// TIA Portal V16 program export: 21 tag tables, 13 data types, 28 data blocks, 76 code blocks (in call order from the OBs), 69 instance data blocks

VAR_GLOBAL   // PLC tag table "Default tag table"
   System_Byte AT %MB1 : Byte;
   FirstScan AT %M1.0 : Bool;
   DiagStatusUpdate AT %M1.1 : Bool;
   AlwaysTRUE AT %M1.2 : Bool;
   AlwaysFALSE AT %M1.3 : Bool;
   Clock_Byte AT %MB0 : Byte;
   Clock_10Hz AT %M0.0 : Bool;
   Clock_5Hz AT %M0.1 : Bool;
   "Clock_2.5Hz" AT %M0.2 : Bool;
   Clock_2Hz AT %M0.3 : Bool;
   "Clock_1.25Hz" AT %M0.4 : Bool;
   Clock_1Hz AT %M0.5 : Bool;
   "Clock_0.625Hz" AT %M0.6 : Bool;
   "Clock_0.5Hz" AT %M0.7 : Bool;
   trig_ustaw_czas AT %M206.1 : Bool;
   trig_pobierz_czas AT %M206.3 : Bool;
   "Bit_6-Wekt-Valve01_R" AT %M2000.6 : Bool;   // Bit-6 kasowanie alarmu
   "Bit_7-Wekt-Valve01_R" AT %M2000.7 : Bool;   // Bit trybu pracy napędu
   "Bit_5-Wekt-Valve01_R" AT %M2000.5 : Bool;   // Rozkaz zamykania
   "Bit_4-Wek_Valve01_R" AT %M2000.4 : Bool;   // Rozkaz otwieranie
   "Bit_0-Wekt_Valve01_R" AT %M2000.0 : Bool;   // Bit gotowośći / awarii
   "Bit_0-Wekt_Valve01_L" AT %M2001.0 : Bool;   // Bit Alarm/Gotowość (Alarm-=1, gotowość=0)
   "Bit_1-Wekt_Valve01_L" AT %M2001.1 : Bool;   // Bit potwierdzenia otwarcia
   "Bit_2-Wekt_Valve01_L" AT %M2001.2 : Bool;   // Bit wyboru trybu Zdalne=1 Remontowe=0
   "Bit_3-Wek_Valve01_L" AT %M2001.3 : Bool;   // Bit potwierdzenia zamknięcia
   "Bit_4-Wek_Valve01_L" AT %M2001.4 : Bool;   // Bit rozkazu na otwieranie
   "Bit_5-Wekt-Valve01_L" AT %M2001.5 : Bool;   // Bit rozkazu na zamykanie
   "Bit_6-Wekt-Valve01_L" AT %M2001.6 : Bool;   // Bit kasowania
   "Bit_7-Wekt-Valve01_L" AT %M2001.7 : Bool;   // Bit rodzaju sterowania aut =1 /manual= 0
   Byte_Wekt_Valve01_L AT %MB2001 : Byte;   // Lewy byte wektora napędu
   Byte_Wekt_Valve01_R AT %MB2000 : Byte;   // Prawy byte wektora napędu
   "I0.3" AT %I0.3 : Bool;
   "I0.4" AT %I0.4 : Bool;
   "I0.5" AT %I0.5 : Bool;
   "I0.6" AT %I0.6 : Bool;
   "Q0.3" AT %Q0.3 : Bool;
   "Q0.4" AT %Q0.4 : Bool;
   "Q0.5" AT %Q0.5 : Bool;
   "I6.4" AT %I6.4 : Bool;
   "I6.3" AT %I6.3 : Bool;
   "I6.2" AT %I6.2 : Bool;
   "I9.5" AT %I9.5 : Bool;
   "I9.6" AT %I9.6 : Bool;
   "I9.7" AT %I9.7 : Bool;
   "I3.1" AT %I3.1 : Bool;
   "I3.2" AT %I3.2 : Bool;
   "I3.3" AT %I3.3 : Bool;
   "I3.4" AT %I3.4 : Bool;
   "Q2.5" AT %Q2.5 : Bool;
   "Q2.6" AT %Q2.6 : Bool;
   "Q2.7" AT %Q2.7 : Bool;
   "I6.1" AT %I6.1 : Bool;
   "Bit_1-Wekt_Valve01_R" AT %M2000.1 : Bool;   // Bit potwierdzenia otwarcia
   "Byte_Wekt_POSITION_R(1)" AT %MB2002 : Byte;   // Prawy byte wektora napędu
   "Bit_0-Wekt_POSITION_R(1)" AT %M2002.0 : Bool;   // Bit gotowośći / awarii
   "Bit_1-Wekt_POSITION_R(1)" AT %M2002.1 : Bool;   // Bit potwierdzenia otwarcia
   "Bit_4-Wek_POSITION_R(1)" AT %M2002.4 : Bool;   // Rozkaz otwieranie
   "Bit_5-Wekt_POSITION_R(1)" AT %M2002.5 : Bool;   // Rozkaz zamykania
   "Bit_6-Wekt_POSITION_R(1)" AT %M2002.6 : Bool;   // Bit-6 kasowanie alarmu
   "Bit_7-Wekt_POSITION_R(1)" AT %M2002.7 : Bool;   // Bit trybu pracy napędu
   "Byte_Wekt_POSITION_L(1)" AT %MB2003 : Byte;   // Lewy byte wektora napędu
   "Bit_0-Wekt_POSITION_L(1)" AT %M2003.0 : Bool;   // Bit Alarm/Gotowość (Alarm-=1, gotowość=0)
   "Bit_1-Wekt_POSITION_L(1)" AT %M2003.1 : Bool;   // Bit potwierdzenia otwarcia
   "Bit_2-Wekt_POSITION_L(1)" AT %M2003.2 : Bool;   // Bit wyboru trybu Zdalne=1 Remontowe=0
   "Bit_3-Wek_POSITION_L(1)" AT %M2003.3 : Bool;   // Bit potwierdzenia zamknięcia
   "Bit_4-Wek_POSITION_L(1)" AT %M2003.4 : Bool;   // Bit rozkazu na otwieranie
   "Bit_5-Wekt_POSITION_L(1)" AT %M2003.5 : Bool;   // Bit rozkazu na zamykanie
   "Bit_6-Wekt_POSITION_L(1)" AT %M2003.6 : Bool;   // Bit kasowania
   "Bit_7-Wekt_POSITION_L(1)" AT %M2003.7 : Bool;   // Bit rodzaju sterowania aut =1 /manual= 0
   "Bit_2-Wekt_POSITION_R(1)" AT %M2002.2 : Bool;   // Bit wyboru trybu Zdalne=1 Remontowe=0
   "Bit_3-Wek_POSITION_R(1)" AT %M2002.3 : Bool;   // Bit potwierdzenia zamknięcia
   Tag_1 AT %M5000.0 : Bool;
   Tag_2 AT %M5000.1 : Bool;
   Tag_3 AT %M5000.3 : Bool;
   "I3.6" AT %I3.6 : Bool;
   "I3.7" AT %I3.7 : Bool;
   "I4.0" AT %I4.0 : Bool;
   "I3.5" AT %I3.5 : Bool;
   "I6.7" AT %I6.7 : Bool;
   "I6.6" AT %I6.6 : Bool;
   "I6.5" AT %I6.5 : Bool;
   "Q3.0" AT %Q3.0 : Bool;
   "Q3.1" AT %Q3.1 : Bool;
   "Q3.2" AT %Q3.2 : Bool;
   My_1Hz AT %M206.7 : Bool;
   "I1.1" AT %I1.1 : Bool;
   "I0.7" AT %I0.7 : Bool;
   "I1.0" AT %I1.0 : Bool;
   "I1.2" AT %I1.2 : Bool;
   "I7.0" AT %I7.0 : Bool;
   "I7.1" AT %I71.1 : Bool;
   "I7.2" AT %I7.2 : Bool;
   "Q3.4" AT %Q3.4 : Bool;
   "Q3.5" AT %Q3.5 : Bool;
   "Q3.6" AT %Q3.6 : Bool;
   "Q1.1" AT %Q1.1 : Bool;
   "Q2.0" AT %Q2.0 : Bool;
   "Q2.1" AT %Q2.1 : Bool;
   "I1.3" AT %I1.3 : Bool;
   "I1.4" AT %I1.4 : Bool;
   "I1.5" AT %I1.5 : Bool;
   "I2.0" AT %I2.0 : Bool;
   "I7.6" AT %I7.6 : Bool;
   "I7.7" AT %I7.7 : Bool;
   "I8.0" AT %I8.0 : Bool;
   "I7.3" AT %I7.3 : Bool;
   "I7.4" AT %I7.4 : Bool;
   "I7.5" AT %I7.5 : Bool;
   "I4.1" AT %I4.1 : Bool;
   "I4.2" AT %I4.2 : Bool;
   "I4.3" AT %I4.3 : Bool;
   "I4.4" AT %I4.4 : Bool;
   "I8.1" AT %I8.1 : Bool;
   "I8.2" AT %I8.2 : Bool;
   "I8.3" AT %I8.3 : Bool;
   "I4.5" AT %I4.5 : Bool;
   "I4.6" AT %I4.6 : Bool;
   "I4.7" AT %I4.7 : Bool;
   "I5.0" AT %I5.0 : Bool;
   "Q3.7" AT %Q3.7 : Bool;
   "Q4.0" AT %Q4.0 : Bool;
   "Q4.1" AT %Q4.1 : Bool;
   "Q2.2" AT %Q2.2 : Bool;
   "Q2.3" AT %Q2.3 : Bool;
   "Q2.4" AT %Q2.4 : Bool;
   "I2.1" AT %I2.1 : Bool;
   "I2.2" AT %I2.2 : Bool;
   "I2.3" AT %I2.3 : Bool;
   "I2.4" AT %I2.4 : Bool;
   "I8.4" AT %I8.4 : Bool;
   "I8.5" AT %I8.5 : Bool;
   "I8.6" AT %I8.6 : Bool;
   "I8.7" AT %I8.7 : Bool;
   "I9.0" AT %I9.0 : Bool;
   "I9.1" AT %I9.1 : Bool;
   "I5.1" AT %I5.1 : Bool;
   "I5.2" AT %I5.2 : Bool;
   "I5.3" AT %I5.3 : Bool;
   "I5.4" AT %I5.4 : Bool;
   "Q4.2" AT %Q4.2 : Bool;
   "Q4.3" AT %Q4.3 : Bool;
   "Q4.4" AT %Q4.4 : Bool;
   "I9.2" AT %I9.2 : Bool;
   "I9.3" AT %I9.3 : Bool;
   "I9.4" AT %I9.4 : Bool;
   "I0.0" AT %I0.0 : Bool;
   "I0.1" AT %I0.1 : Bool;
   "I0.2" AT %I0.2 : Bool;
   "Q0.6" AT %Q0.6 : Bool;
   "Q0.7" AT %Q0.7 : Bool;
   "Q1.0" AT %Q1.0 : Bool;
   "Q0.0" AT %Q0.0 : Bool;
   "Q0.1" AT %Q0.1 : Bool;
   "Q0.2" AT %Q0.2 : Bool;
   "I10.0" AT %I10.0 : Bool;
   setTime AT %M8.0 : Bool;   // ustaw zegar
   setData AT %M8.1 : Bool;   // ustaw datę
   isDaily AT %M80.7 : Bool;   // tryb sterowania dobowy
   isWeekiy AT %M81.0 : Bool;   // tryb sterowania tygodniowy
   isPowerOK AT %M81.2 : Bool;   // znacznik powrotu zasilania
   Tag_4 AT %Q6.7 : Bool;
   zbocze_dod_zegar AT %M47.0 : Bool;
   ResetErrorOB82 AT %M91.1 : Bool;
   "I5.5" AT %I5.5 : Bool;
   "I5.6" AT %I5.6 : Bool;
   "I5.7" AT %I5.7 : Bool;
   "I6.0" AT %I6.0 : Bool;
END_VAR
VAR_GLOBAL CONSTANT   // user constants
   analog_error_H : Word := 28538;
   CONST_BUFFER_OB82 : USInt := 200;
END_VAR

VAR_GLOBAL   // PLC tag table "Alarm_error"
   errorAnlog_Z10 AT %M9.3 : Bool;   // sygnał błędu sygnału analogowego położenia Z10
   outAlarm AT %M1030.3 : Bool;   // Znacznik alarmu zbiorczego (Sygnalizator)
   float_min_tank_4 AT %M47.4 : Bool;   // pływak min zbiornik 4
   float_min_tank_1 AT %M47.1 : Bool;   // pływak min zbiornik 1
   float_min_tank_3 AT %M47.3 : Bool;   // pływak min zbiornik 3
   float_min_tank_2 AT %M47.2 : Bool;   // pływak min zbiornik 2
   "I2.7" AT %I2.7 : Bool;
   "I3.0" AT %I3.0 : Bool;
   "I2.6" AT %I2.6 : Bool;
   "I2.5" AT %I2.5 : Bool;
   Communication_alarm_tcp AT %M1030.2 : Bool;   // Znacznik błedu komunikacji HMI - PLC
   comunication_alarm_modbus_rtu AT %M1030.4 : Bool;   // kontrola przebiegu pętli odczytu parametró z modbus rtu
   Led_Error AT %M91.0 : Bool;   // bit sygnalizacji zapalenia led error na CPU
   Status_QRY AT %MW302 : Word;   // Status słowa przerwań (bit 0 - informacja o CPU 0- RUN, 1- Rozruch)
   statusCPU AT %M302.0 : Bool;   // 0- Run 1-Rozruch
   Error_QRY AT %MW300 : Int;   // Słowo błędu przetwarzania przerwań czasowych
   setAlarmNiskie_magistrala AT %M91.2 : Bool;   // bit alarmu niskiego ciśnienia na magistrali
   resetAlarmNiskie_magistrala AT %M91.3 : Bool;   // bit końca niskiego ciśnienia magistrala
   float_max_tank_3 AT %M46.6 : Bool;   // pływak max zbiornik 3
   float_max_tank_1 AT %M46.4 : Bool;   // pływak max zbiornik 1
   setControl_alarm_B5 AT %M91.4 : Bool;   // Załczenie sterowania zbiornikami w trybie awarii na magistrali
   float_max_tank_2 AT %M46.5 : Bool;   // pływak max zbiornik 2
   float_max_tank_4 AT %M46.7 : Bool;   // pływak max zbiornik 2
   reset_error_hwork AT %M45.6 : Bool;   // reset po błędzie gdy wszystkie zbiorniki ten sam czas pracy
END_VAR

VAR_GLOBAL   // PLC tag table "Analogi"
   AI_poziom_zbiornik_4 AT %MW42 : Word;
   AI_poziom_zbiornik_2 AT %MW38 : Word;
   IW68 AT %IW68 : Word;   // wejscie AI
   AI_poziom_zbiornik_1 AT %MW36 : Word;
   AI_poziom_zbiornik_3 AT %MW40 : Word;
   IW78 AT %IW78 : Word;   // wejscie AI
   AI_położenie_Z10 AT %MW34 : Word;
   AI_przepływ AT %MW30 : Word;
   AI_ciśnienie_B5 AT %MW32 : Word;
   IW70 AT %IW70 : Word;   // wejscie AI
   IW72 AT %IW72 : Word;   // wejscie AI
   IW76 AT %IW76 : Word;   // wejscie AI
   IW74 AT %IW74 : Word;   // wejscie AI
   switch_Kolman AT %M46.0 : Bool;   // przełącznik funkcji filtr analogów (Kolman = OFF, bez Kolman = ON)
   I AT %MW48 : Int;   // kalman zmienna przechwuje adres wejścia AI
END_VAR

VAR_GLOBAL   // PLC tag table "Tag HMI"
   "HMI.ManualMode_visible" AT %M1023.1 : Bool;
   "HMI.ErrorBits_Int" AT %MW1024 : Int;
   "HMI.Warning_Int" AT %MW1028 : Int;
   "HMI.ErrorAck_Int" AT %MW1026 : Int;
   ProcessMemory_Static_1_setChanging AT %M9.2 : Bool;   // Znacznik pobierania konfiguracji do instancji pamięci peocesu
   "HMI.Acknowledge_visible" AT %M1030.1 : Bool;
   memRis_WatchDog_HMI_PLC AT %M9.0 : Bool;
   "HMI.ErrorAck" AT %M1030.0 : Bool;
   "HMI.Filing3" AT %M1031.4 : Bool;   // bit informujący o wejściu w tryb napełniania
   "HMI.Warning_Int_tank" AT %MW1031 : Int;
   "HMI.rez" AT %M1031.1 : Bool;
   "HMI.StopFiling" AT %M1031.0 : Bool;   // bit informacji o zatrzymanym napełnianiu z powodu niskiego ciśnienia wna magistrali
   "HMI.Filing2" AT %M1031.3 : Bool;   // bit informujący o wejściu w tryb napełniania
   "HMI.Filing4" AT %M1031.5 : Bool;   // bit informujący o wejściu w tryb napełniania
   "HMI.Filing1" AT %M1031.2 : Bool;   // bit informujący o wejściu w tryb napełniania
END_VAR

VAR_GLOBAL   // PLC tag table "ModbusRTU"
   switch_flow_analog_modbus AT %M79.0 : Bool;   // przełącznik wyboru medium pomiaru przepływu z wy analogowego czy modbus rtu
END_VAR

VAR_GLOBAL   // PLC tag table "ModbusTCP"
   memTrig_Client_ReceivingTIME AT %M206.4 : Bool;
   memTrig_Step_Sending AT %M9.4 : Bool;   // Pamieć zbocza na uruchomienie pętli Modbus TCP wysyłanie
   done_modbusTCP_przetworzone AT %M9.1 : Bool;   // bit zezwala na wysłanie danych po przetworzeniu przez program PLC Zasuwy
   memTrig_Step_Receiving_Time AT %M9.6 : Bool;   // Pamieć zbocza na uruchomienie pętli Modbus TCP pobieranie Time
   memTrig_Step_Receiving AT %M9.5 : Bool;   // Pamieć zbocza na uruchomienie pętli Modbus TCP pobieranie
   memRisingTriger_Data_13 AT %M208.4 : Bool;   // pamieć zbocza zmiany danych w zmiennej
   memRisingTriger_Data_9 AT %M208.0 : Bool;   // pamieć zbocza zmiany danych w zmiennej
   memRisingTriger_Data_6 AT %M207.5 : Bool;   // pamieć zbocza zmiany danych w zmiennej
   memRisingTriger_Data_5 AT %M207.4 : Bool;   // pamieć zbocza zmiany danych w zmiennej
   memRisingTriger_Data_7 AT %M207.6 : Bool;   // pamieć zbocza zmiany danych w zmiennej
   memRisingTriger_Data_10 AT %M208.1 : Bool;   // pamieć zbocza zmiany danych w zmiennej
   memRisingTriger_Data_8 AT %M207.7 : Bool;   // pamieć zbocza zmiany danych w zmiennej
   memRisingTriger_Data_11 AT %M208.2 : Bool;   // pamieć zbocza zmiany danych w zmiennej
   memRisingTriger_Data_1 AT %M207.0 : Bool;   // pamieć zbocza zmiany danych w zmiennej
   memRisingTriger_Data_2 AT %M207.1 : Bool;   // pamieć zbocza zmiany danych w zmiennej
   memRisingTriger_Data_4 AT %M207.3 : Bool;   // pamieć zbocza zmiany danych w zmiennej
   memRisingTriger_Data_12 AT %M208.3 : Bool;   // pamieć zbocza zmiany danych w zmiennej
   memRisingTriger_Data_3 AT %M207.2 : Bool;   // pamieć zbocza zmiany danych w zmiennej
   memRisingTriger_Data_1_2 AT %M212.4 : Bool;   // pamieć zbocza zmiany danych w zmiennej
   memTrig_SendingError_4 AT %M210.7 : Bool;   // bit pamęci zbocza błedu wysyłania modbus tCP
   memTrig_Client_Receiving_12 AT %M210.1 : Bool;   // pamieć zbocza zmiany danych w zmiennej
   memTrig_Client_Receiving_3 AT %M209.0 : Bool;   // pamieć zbocza zmiany danych w zmiennej
   memTrig_Client_Receiving_9 AT %M209.6 : Bool;   // pamieć zbocza zmiany danych w zmiennej
   memTrig_Client_Receiving_11 AT %M210.0 : Bool;   // pamieć zbocza zmiany danych w zmiennej
   memTrig_Step_Sending_1 AT %M211.0 : Bool;   // Pamieć zbocza na uruchomienie pętli Modbus TCP wysyłanie
   memTrig_Client_Receiving_6 AT %M209.3 : Bool;   // pamieć zbocza zmiany danych w zmiennej
   memTrig_Client_Receiving_4 AT %M209.1 : Bool;   // pamieć zbocza zmiany danych w zmiennej
   done_modbusTCP_przetw_1 AT %M211.1 : Bool;   // bit zezwala na wysłanie danych po przetworzeniu przez program PLC Zasuwy
   memTrig_SendingError_2 AT %M210.5 : Bool;   // bit pamęci zbocza błedu wysyłania modbus tCP
   done_modbusTCP_przetw_6 AT %M212.2 : Bool;   // bit zezwala na wysłanie danych po przetworzeniu przez program PLC Zasuwy
   memTrig_Client_Receiving_2 AT %M208.7 : Bool;   // pamieć zbocza zmiany danych w zmiennej
   done_modbusTCP_przetw_4 AT %M212.0 : Bool;   // bit zezwala na wysłanie danych po przetworzeniu przez program PLC Zasuwy
   done_modbusTCP_przetw_2 AT %M211.2 : Bool;   // bit zezwala na wysłanie danych po przetworzeniu przez program PLC Zasuwy
   memTrig_Client_Receiving_7 AT %M209.4 : Bool;   // pamieć zbocza zmiany danych w zmiennej
   memTrig_Client_Receiving_13 AT %M210.2 : Bool;   // pamieć zbocza zmiany danych w zmiennej
   memRisingTriger_Data_1_1 AT %M212.3 : Bool;   // pamieć zbocza zmiany danych w zmiennej
   memTrig_Client_Receiving_5 AT %M209.2 : Bool;   // pamieć zbocza zmiany danych w zmiennej
   memRisingTriger_Data_1_5 AT %M212.7 : Bool;   // pamieć zbocza zmiany danych w zmiennej
   memTrig_Client_Receiving_1 AT %M208.6 : Bool;   // pamieć zbocza zmiany danych w zmiennej
   memTrig_Step_Sending_4 AT %M211.6 : Bool;   // Pamieć zbocza na uruchomienie pętli Modbus TCP wysyłanie
   memTrig_Client_Receiving_10 AT %M209.7 : Bool;   // pamieć zbocza zmiany danych w zmiennej
   memRisingTriger_Data_1_4 AT %M212.6 : Bool;   // pamieć zbocza zmiany danych w zmiennej
   memTrig_Client_Receiving_8 AT %M209.5 : Bool;   // pamieć zbocza zmiany danych w zmiennej
   memTrig_SendingError_3 AT %M210.6 : Bool;   // bit pamęci zbocza błedu wysyłania modbus tCP
   memTrig_Step_Sending_5 AT %M211.7 : Bool;   // Pamieć zbocza na uruchomienie pętli Modbus TCP wysyłanie
   done_modbusTCP_przetw_3 AT %M211.3 : Bool;   // bit zezwala na wysłanie danych po przetworzeniu przez program PLC Zasuwy
   memRisingTriger_Data_1_3 AT %M212.5 : Bool;   // pamieć zbocza zmiany danych w zmiennej
   memTrig_Step_Sending_2 AT %M211.4 : Bool;   // Pamieć zbocza na uruchomienie pętli Modbus TCP wysyłanie
   done_modbusTCP_przetw_5 AT %M212.1 : Bool;   // bit zezwala na wysłanie danych po przetworzeniu przez program PLC Zasuwy
   memTrig_SendingError_1 AT %M210.4 : Bool;   // bit pamęci zbocza błedu wysyłania modbus tCP
   memTrig_Client_Receiving_14 AT %M210.3 : Bool;   // pamieć zbocza zmiany danych w zmiennej
   memTrig_Step_Sending_3 AT %M211.5 : Bool;   // Pamieć zbocza na uruchomienie pętli Modbus TCP wysyłanie
   memTrig_Error_Receiving AT %M208.5 : Bool;   // pamieć zboczawystąpienia błędu pobierania
   memRisingTriger_Data_16 AT %M213.2 : Bool;   // pamieć zbocza zmiany danych w zmiennej
   memTrig_Client_Receiving_15 AT %M213.3 : Bool;   // pamieć zbocza zmiany danych w zmiennej
   memRisingTriger_Data_14 AT %M213.0 : Bool;   // pamieć zbocza zmiany danych w zmiennej
   memTrig_Client_Receiving_16 AT %M213.4 : Bool;   // pamieć zbocza zmiany danych w zmiennej
   memRisingTriger_Data_15 AT %M213.1 : Bool;   // pamieć zbocza zmiany danych w zmiennej
   memTrig_loop_error AT %M206.5 : Bool;   // błąd petli Modbus TCP brak obiegu pętli
   memRisingTriger_Data_50 AT %M227.1 : Bool;
   memTrig_Client_Receiving_37 AT %M216.4 : Bool;   // pamieć zbocza zmiany danych w zmiennej
   memRisingTriger_Data_83 AT %M231.2 : Bool;
   memTrig_Client_Receiving_84 AT %M222.3 : Bool;   // pamieć zbocza zmiany danych w zmiennej
   memRisingTriger_Data_76 AT %M230.3 : Bool;
   memRisingTriger_Data_18 AT %M223.1 : Bool;
   memTrig_Client_Receiving_38 AT %M216.5 : Bool;   // pamieć zbocza zmiany danych w zmiennej
   memRisingTriger_Data_89 AT %M232.0 : Bool;
   memTrig_Client_Receiving_17 AT %M214.0 : Bool;   // pamieć zbocza zmiany danych w zmiennej
   memTrig_Client_Receiving_81 AT %M222.0 : Bool;   // pamieć zbocza zmiany danych w zmiennej
   memRisingTriger_Data_81 AT %M231.0 : Bool;
   memTrig_Client_Receiving_66 AT %M220.1 : Bool;   // pamieć zbocza zmiany danych w zmiennej
   memTrig_Client_Receiving_62 AT %M219.5 : Bool;   // pamieć zbocza zmiany danych w zmiennej
   memTrig_Client_Receiving_21 AT %M214.4 : Bool;   // pamieć zbocza zmiany danych w zmiennej
   memTrig_Client_Receiving_65 AT %M220.0 : Bool;   // pamieć zbocza zmiany danych w zmiennej
   memTrig_Client_Receiving_43 AT %M217.2 : Bool;   // pamieć zbocza zmiany danych w zmiennej
   memRisingTriger_Data_85 AT %M231.4 : Bool;
   memTrig_Client_Receiving_25 AT %M215.0 : Bool;   // pamieć zbocza zmiany danych w zmiennej
   memRisingTriger_Data_70 AT %M229.5 : Bool;
   memTrig_Client_Receiving_46 AT %M217.5 : Bool;   // pamieć zbocza zmiany danych w zmiennej
   memTrig_Client_Receiving_47 AT %M217.6 : Bool;   // pamieć zbocza zmiany danych w zmiennej
   memTrig_Client_Receiving_18 AT %M214.1 : Bool;   // pamieć zbocza zmiany danych w zmiennej
   memRisingTriger_Data_40 AT %M225.7 : Bool;
   memRisingTriger_Data_86 AT %M231.5 : Bool;
   memRisingTriger_Data_68 AT %M229.3 : Bool;
   memTrig_Client_Receiving_19 AT %M214.2 : Bool;   // pamieć zbocza zmiany danych w zmiennej
   memTrig_Client_Receiving_41 AT %M217.0 : Bool;   // pamieć zbocza zmiany danych w zmiennej
   memRisingTriger_Data_45 AT %M226.4 : Bool;
   memTrig_Client_Receiving_64 AT %M219.7 : Bool;   // pamieć zbocza zmiany danych w zmiennej
   memRisingTriger_Data_28 AT %M224.3 : Bool;
   memTrig_Client_Receiving_49 AT %M218.0 : Bool;   // pamieć zbocza zmiany danych w zmiennej
   memRisingTriger_Data_65 AT %M229.0 : Bool;
   memTrig_Client_Receiving_35 AT %M216.2 : Bool;   // pamieć zbocza zmiany danych w zmiennej
   memRisingTriger_Data_21 AT %M223.4 : Bool;
   memTrig_Client_Receiving_72 AT %M220.7 : Bool;   // pamieć zbocza zmiany danych w zmiennej
   memTrig_Client_Receiving_57 AT %M219.0 : Bool;   // pamieć zbocza zmiany danych w zmiennej
   memTrig_Client_Receiving_51 AT %M218.2 : Bool;   // pamieć zbocza zmiany danych w zmiennej
   memTrig_Client_Receiving_28 AT %M215.3 : Bool;   // pamieć zbocza zmiany danych w zmiennej
   memRisingTriger_Data_66 AT %M229.1 : Bool;
   memTrig_Client_Receiving_45 AT %M217.4 : Bool;   // pamieć zbocza zmiany danych w zmiennej
   memTrig_Client_Receiving_89 AT %M223.0 : Bool;   // pamieć zbocza zmiany danych w zmiennej
   memRisingTriger_Data_35 AT %M225.2 : Bool;
   memTrig_Client_Receiving_83 AT %M222.2 : Bool;   // pamieć zbocza zmiany danych w zmiennej
   memRisingTriger_Data_56 AT %M227.7 : Bool;
   memRisingTriger_Data_20 AT %M223.3 : Bool;
   memTrig_Client_Receiving_36 AT %M216.3 : Bool;   // pamieć zbocza zmiany danych w zmiennej
   memTrig_Client_Receiving_26 AT %M215.1 : Bool;   // pamieć zbocza zmiany danych w zmiennej
   memRisingTriger_Data_23 AT %M223.6 : Bool;
   memRisingTriger_Data_48 AT %M226.7 : Bool;
   memRisingTriger_Data_64 AT %M228.7 : Bool;
   memRisingTriger_Data_61 AT %M228.4 : Bool;
   memRisingTriger_Data_36 AT %M225.3 : Bool;
   memRisingTriger_Data_88 AT %M231.7 : Bool;
   memTrig_Client_Receiving_76 AT %M221.3 : Bool;   // pamieć zbocza zmiany danych w zmiennej
   memRisingTriger_Data_72 AT %M229.7 : Bool;
   memRisingTriger_Data_74 AT %M230.1 : Bool;
   memRisingTriger_Data_39 AT %M225.6 : Bool;
   memRisingTriger_Data_90 AT %M232.1 : Bool;
   memRisingTriger_Data_25 AT %M224.0 : Bool;
   memRisingTriger_Data_44 AT %M226.3 : Bool;
   memRisingTriger_Data_80 AT %M230.7 : Bool;
   memTrig_Client_Receiving_70 AT %M220.5 : Bool;   // pamieć zbocza zmiany danych w zmiennej
   memRisingTriger_Data_37 AT %M225.4 : Bool;
   memTrig_Client_Receiving_20 AT %M214.3 : Bool;   // pamieć zbocza zmiany danych w zmiennej
   memTrig_Client_Receiving_34 AT %M216.1 : Bool;   // pamieć zbocza zmiany danych w zmiennej
   memRisingTriger_Data_49 AT %M227.0 : Bool;
   memRisingTriger_Data_78 AT %M230.5 : Bool;
   memRisingTriger_Data_38 AT %M225.5 : Bool;
   memTrig_Client_Receiving_87 AT %M222.6 : Bool;   // pamieć zbocza zmiany danych w zmiennej
   memTrig_Client_Receiving_30 AT %M215.5 : Bool;   // pamieć zbocza zmiany danych w zmiennej
   memRisingTriger_Data_42 AT %M226.1 : Bool;
   memRisingTriger_Data_57 AT %M228.0 : Bool;
   memTrig_Client_Receiving_54 AT %M218.5 : Bool;   // pamieć zbocza zmiany danych w zmiennej
   memRisingTriger_Data_77 AT %M230.4 : Bool;
   memTrig_Client_Receiving_86 AT %M222.5 : Bool;   // pamieć zbocza zmiany danych w zmiennej
   memTrig_Client_Receiving_63 AT %M219.6 : Bool;   // pamieć zbocza zmiany danych w zmiennej
   memTrig_Client_Receiving_67 AT %M220.2 : Bool;   // pamieć zbocza zmiany danych w zmiennej
   memTrig_Client_Receiving_75 AT %M221.2 : Bool;   // pamieć zbocza zmiany danych w zmiennej
   memRisingTriger_Data_54 AT %M227.5 : Bool;
   memTrig_Client_Receiving_24 AT %M214.7 : Bool;   // pamieć zbocza zmiany danych w zmiennej
   memRisingTriger_Data_41 AT %M226.0 : Bool;
   memTrig_Client_Receiving_82 AT %M222.1 : Bool;   // pamieć zbocza zmiany danych w zmiennej
   memRisingTriger_Data_75 AT %M230.2 : Bool;
   memTrig_Client_Receiving_61 AT %M219.4 : Bool;   // pamieć zbocza zmiany danych w zmiennej
   memRisingTriger_Data_59 AT %M228.2 : Bool;
   memRisingTriger_Data_33 AT %M225.0 : Bool;
   memRisingTriger_Data_19 AT %M223.2 : Bool;
   memTrig_Client_Receiving_56 AT %M218.7 : Bool;   // pamieć zbocza zmiany danych w zmiennej
   memTrig_Client_Receiving_88 AT %M222.7 : Bool;   // pamieć zbocza zmiany danych w zmiennej
   memRisingTriger_Data_47 AT %M226.6 : Bool;
   memTrig_Client_Receiving_59 AT %M219.2 : Bool;   // pamieć zbocza zmiany danych w zmiennej
   memTrig_Client_Receiving_48 AT %M217.7 : Bool;   // pamieć zbocza zmiany danych w zmiennej
   memTrig_Client_Receiving_23 AT %M214.6 : Bool;   // pamieć zbocza zmiany danych w zmiennej
   memTrig_Client_Receiving_32 AT %M215.7 : Bool;   // pamieć zbocza zmiany danych w zmiennej
   memTrig_Client_Receiving_53 AT %M218.4 : Bool;   // pamieć zbocza zmiany danych w zmiennej
   memRisingTriger_Data_79 AT %M230.6 : Bool;
   memRisingTriger_Data_43 AT %M226.2 : Bool;
   memRisingTriger_Data_73 AT %M230.0 : Bool;
   memRisingTriger_Data_87 AT %M231.6 : Bool;
   memRisingTriger_Data_58 AT %M228.1 : Bool;
   memRisingTriger_Data_69 AT %M229.4 : Bool;
   memTrig_Client_Receiving_42 AT %M217.1 : Bool;   // pamieć zbocza zmiany danych w zmiennej
   memTrig_Client_Receiving_69 AT %M220.4 : Bool;   // pamieć zbocza zmiany danych w zmiennej
   memTrig_Client_Receiving_44 AT %M217.3 : Bool;   // pamieć zbocza zmiany danych w zmiennej
   memTrig_Client_Receiving_85 AT %M222.4 : Bool;   // pamieć zbocza zmiany danych w zmiennej
   memTrig_Client_Receiving_31 AT %M215.6 : Bool;   // pamieć zbocza zmiany danych w zmiennej
   memTrig_Client_Receiving_27 AT %M215.2 : Bool;   // pamieć zbocza zmiany danych w zmiennej
   memRisingTriger_Data_24 AT %M223.7 : Bool;
   memTrig_Client_Receiving_50 AT %M218.1 : Bool;   // pamieć zbocza zmiany danych w zmiennej
   memRisingTriger_Data_17 AT %M206.6 : Bool;
   memTrig_Client_Receiving_22 AT %M214.5 : Bool;   // pamieć zbocza zmiany danych w zmiennej
   memRisingTriger_Data_52 AT %M227.3 : Bool;
   memRisingTriger_Data_55 AT %M227.6 : Bool;
   memRisingTriger_Data_34 AT %M225.1 : Bool;
   memTrig_Client_Receiving_77 AT %M221.4 : Bool;   // pamieć zbocza zmiany danych w zmiennej
   memRisingTriger_Data_82 AT %M231.1 : Bool;
   memRisingTriger_Data_67 AT %M229.2 : Bool;
   memRisingTriger_Data_26 AT %M224.1 : Bool;
   memTrig_Client_Receiving_60 AT %M219.3 : Bool;   // pamieć zbocza zmiany danych w zmiennej
   memRisingTriger_Data_27 AT %M224.2 : Bool;
   memTrig_Client_Receiving_52 AT %M218.3 : Bool;   // pamieć zbocza zmiany danych w zmiennej
   memRisingTriger_Data_84 AT %M231.3 : Bool;
   memTrig_Client_Receiving_29 AT %M215.4 : Bool;   // pamieć zbocza zmiany danych w zmiennej
   memTrig_Client_Receiving_73 AT %M221.0 : Bool;   // pamieć zbocza zmiany danych w zmiennej
   memRisingTriger_Data_62 AT %M228.5 : Bool;
   memTrig_Client_Receiving_58 AT %M219.1 : Bool;   // pamieć zbocza zmiany danych w zmiennej
   memRisingTriger_Data_71 AT %M229.6 : Bool;
   memTrig_Client_Receiving_79 AT %M221.6 : Bool;   // pamieć zbocza zmiany danych w zmiennej
   memTrig_Client_Receiving_33 AT %M216.0 : Bool;   // pamieć zbocza zmiany danych w zmiennej
   memRisingTriger_Data_22 AT %M223.5 : Bool;
   memTrig_Client_Receiving_74 AT %M221.1 : Bool;   // pamieć zbocza zmiany danych w zmiennej
   memRisingTriger_Data_51 AT %M227.2 : Bool;
   memTrig_Client_Receiving_78 AT %M221.5 : Bool;   // pamieć zbocza zmiany danych w zmiennej
   memTrig_Client_Receiving_55 AT %M218.6 : Bool;   // pamieć zbocza zmiany danych w zmiennej
   memRisingTriger_Data_30 AT %M224.5 : Bool;
   memTrig_Client_Receiving_40 AT %M216.7 : Bool;   // pamieć zbocza zmiany danych w zmiennej
   memRisingTriger_Data_53 AT %M227.4 : Bool;
   memRisingTriger_Data_29 AT %M224.4 : Bool;
   memRisingTriger_Data_32 AT %M224.7 : Bool;
   memRisingTriger_Data_46 AT %M226.5 : Bool;
   memRisingTriger_Data_60 AT %M228.3 : Bool;
   memRisingTriger_tmerDisconected AT %M228.6 : Bool;   // znacznik załączenia opóźnienia
   timerDISCONECTED_TCP_SERVER_1 AT %M216.6 : Bool;   // znacznik opoźnienia rozłączenia tcp modbus
   timerDISCONECTED_TCP_SERVER_2 AT %M220.3 : Bool;   // znacznik opoźnienia rozłączenia tcp modbus
   timerDISCONECTED_TCP_SERVER_3 AT %M220.6 : Bool;   // znacznik opoźnienia rozłączenia tcp modbus
   timerDISCONECTED_TCP_SERVER_4 AT %M221.7 : Bool;   // znacznik opoźnienia rozłączenia tcp modbus
   memRisingTriger_resetModbusTCP AT %M224.6 : Bool;   // znacznik przerwania połaczenia Modbus TCP na 10sek
END_VAR

VAR_GLOBAL   // PLC tag table "RTC"
   "memStep_errorMPP04-2" AT %MB103 : USInt;   // bajt pamieci w którym kroku nastąpił błąd modbus
   setErrorModbsmasterMPP04_2 AT %M104.3 : Bool;   // error bit modbus master przepływomierz / Znacznik błedu komunikacji modbus
   "memRisSteperror_MPP04-2" AT %M104.1 : Bool;   // pamięć zbocza dla przechwycenia kroku błedu
   memRisErrorModbusMPP04_2 AT %M104.2 : Bool;   // pamięć zbocza error modbus MPP04-1
   Pobierz_czas AT %M206.2 : Bool;
   Ustaw_czas AT %M206.0 : Bool;
   status_wr_sys_t AT %MW204 : Int;
   status_rd_loc_t AT %MW202 : Int;
   status_rd_sys_t AT %MW200 : Int;
END_VAR

VAR_GLOBAL   // PLC tag table "Tag Sim"
   Sim_23 AT %M3002.6 : Bool;
   Sim_22 AT %M3002.5 : Bool;
   Sim_21 AT %M3002.4 : Bool;
   Sim_24 AT %M3002.7 : Bool;
   Sim_19 AT %M3002.2 : Bool;
   Sim_generator_reg AT %M3002.3 : Bool;
   Sim__Z5_Open_Spust AT %M3001.1 : Bool;
   Sim__Z2_Colse_Wlot AT %M3000.2 : Bool;
   Sim__Z6_Open_Wlot AT %M3001.3 : Bool;
   Sim__Z1_Open_Spust AT %M3000.1 : Bool;
   Sim__Z1_Close_Spust AT %M3000.0 : Bool;
   Sim__Z6_Close_Wlot AT %M3001.2 : Bool;
   Sim__Z8_Close_Wylot AT %M3001.6 : Bool;
   Sim__Z3_Open_Spust AT %M3000.5 : Bool;
   Sim__Z9_Close AT %M3002.0 : Bool;
   Sim__Z5_Close_Spust AT %M3001.0 : Bool;
   Sim__Z3_Close_Spust AT %M3000.4 : Bool;
   Sim__Z4_Close_Wlot AT %M3000.6 : Bool;
   Sim__Z2_Open_Wlot AT %M3000.3 : Bool;
   Sim__Z9_Open AT %M3002.1 : Bool;
   Sim__Z8_Open_Wlot AT %M3001.7 : Bool;
   Sim__Z4_Open_Wlot AT %M3000.7 : Bool;
   Sim__Z7_Close_Spust AT %M3001.4 : Bool;
   Sim__Z7_Open_Spust AT %M3001.5 : Bool;
   Sim__Z7_TCP_error AT %M3003.0 : Bool;
   Sim__Z10_close AT %M3003.2 : Bool;
   Sim__Z10_open AT %M3003.1 : Bool;
   "auto set open" AT %M3003.3 : Bool;
   "auto set close" AT %M3003.4 : Bool;
END_VAR

VAR_GLOBAL   // PLC tag table "Tag VLV01"
END_VAR

VAR_GLOBAL   // PLC tag table "Z1"
   Hbit_Zamknij_Z1 AT %M10.5 : Bool;
   Hbit_Alarm_Z1 AT %M10.0 : Bool;
   CMD_Awaria_Z_1 AT %M52.0 : Bool;   // Awaria zbiorcza
   inputAumaawariaZ_1 AT %M51.2 : Bool;   // znacznik wejście
   Hbit_Otwarta_Z1 AT %M10.1 : Bool;
   Hbit_Zamknieta_Z1 AT %M10.3 : Bool;
   Byte_Status_Z1 AT %MW10 : Word;   // Słowo statusu napędu
   inputAumagotowośćZ_1 AT %M51.1 : Bool;   // znacznik wejście
   inputAwariaMomentZ_1 AT %M50.6 : Bool;   // znacznik wejście
   isGotowość_Z_1 AT %M50.0 : Bool;   // bit gotowości wspólny
   Hbit_Auto_Manu_Z1 AT %M10.7 : Bool;
   Hbit_Reset_Z1 AT %M10.6 : Bool;
   inputOtwartaZ_1 AT %M50.2 : Bool;   // znacznik wejście
   inputAumalokalneZ_1 AT %M50.7 : Bool;   // znacznik wejście
   setSVMC_Z_1 AT %M51.4 : Bool;   // Znacznik polecenia zamknij w trybie automat
   Hbit_REN_Z1 AT %M10.2 : Bool;
   setAlarm_Moment_Z_1 AT %M51.5 : Bool;   // znacznik alarmu od momentówki w trybie zdalnym (aut/mamnual)
   inputAumaautomatZ_1 AT %M51.0 : Bool;   // znacznik wejście
   inputRuch_Z_1 AT %M50.5 : Bool;   // znacznik wejście
   CMD_Close_Z_1 AT %M51.7 : Bool;   // załącz zamykanie
   inputREMT_Z_1 AT %M50.1 : Bool;   // znacznik wejście zdalne
   CMD_Open_Z_1 AT %M51.6 : Bool;   // załącz otwieranie
   Hbit_Otwórz_Z1 AT %M10.4 : Bool;
   inputZamkniętaZ_1 AT %M50.3 : Bool;   // znacznik wejście
   isAUMA_Z_1 AT %M52.2 : Bool;   // przęłącznik wymiany na AUMA
   setSVMO_Z_1 AT %M51.3 : Bool;   // Znacznik polecenia otwórz w trybie automat
END_VAR

VAR_GLOBAL   // PLC tag table "Z10"
   inputOtwartaZ_10 AT %M72.2 : Bool;   // znacznik wejście
   Hbit_Otwórz_Z10 AT %M28.4 : Bool;
   Hbit_Auto_Manu_Z10 AT %M28.7 : Bool;
   setSVMC_Z_10 AT %M73.3 : Bool;   // Znacznik polecenia zamknij w trybie automat
   setSVMO_Z_10 AT %M73.2 : Bool;   // Znacznik polecenia otwórz w trybie automat
   Hbit_Zamknieta_Z10 AT %M28.3 : Bool;
   setAlarm_Moment_Z_10 AT %M73.4 : Bool;   // znacznik alarmu od momentówki w trybie zdalnym (aut/mamnual)
   inputAumaautomatZ_10 AT %M72.7 : Bool;   // znacznik wejście
   CMD_Close_Z_10 AT %M73.6 : Bool;   // załącz zamykanie
   CMD_Open_Z_10 AT %M73.5 : Bool;   // załącz otwieranie
   inputRuch_Z_10 AT %M72.4 : Bool;   // znacznik wejście
   Byte_Status_Z10 AT %MW28 : Word;   // Słowo statusu napędu
   inputREMT_Z_10 AT %M72.1 : Bool;   // znacznik wejście zdalne
   Hbit_REN_Z10 AT %M28.2 : Bool;
   Hbit_Otwarta_Z10 AT %M28.1 : Bool;
   Hbit_Reset_Z10 AT %M28.6 : Bool;
   inputAumaawariaZ_10 AT %M73.1 : Bool;   // znacznik wejście
   inputAumagotowośćZ_10 AT %M73.0 : Bool;   // znacznik wejście
   Hbit_Zamknij_Z10 AT %M28.5 : Bool;
   CMD_Awaria_Z_10 AT %M73.7 : Bool;   // Awaria zbiorcza
   inputAumalokalneZ_10 AT %M72.6 : Bool;   // znacznik wejście
   isGotowość_Z_10 AT %M72.0 : Bool;   // bit gotowości wspólny
   inputZamkniętaZ_10 AT %M72.3 : Bool;   // znacznik wejście
   Hbit_Alarm_Z10 AT %M28.0 : Bool;
   isOpen_Z10 AT %M52.3 : Bool;   // bit potwierdzenia otwarcia prz sterowaniu [%]
   inputAwariaMomentZ_10 AT %M72.5 : Bool;   // znacznik wejście
   isClose_od_położenia AT %M74.0 : Bool;   // gdy brak sygnały a krancowego wyłacznika to patrzy na pozycję z nadajnika
END_VAR

VAR_GLOBAL   // PLC tag table "Z2"
   Hbit_Reset_Z2 AT %M12.6 : Bool;
   inputREMT_Z_2 AT %M53.1 : Bool;   // znacznik wejście zdalne
   Hbit_Zamknij_Z2 AT %M12.5 : Bool;
   Hbit_Otwarta_Z2 AT %M12.1 : Bool;
   Byte_Status_Z2 AT %MW12 : Word;   // Słowo statusu napędu
   inputAwariaMomentZ_2 AT %M53.5 : Bool;   // znacznik wejście
   inputZamkniętaZ_2 AT %M53.3 : Bool;   // znacznik wejście
   Hbit_Alarm_Z2 AT %M12.0 : Bool;
   Hbit_Zamknieta_Z2 AT %M12.3 : Bool;
   inputRuch_Z_2 AT %M53.4 : Bool;
   setSVMC_Z_2 AT %M54.3 : Bool;   // Znacznik polecenia zamknij w trybie automat
   inputAumalokalneZ_2 AT %M53.6 : Bool;   // znacznik wejście
   Hbit_Auto_Manu_Z2 AT %M12.7 : Bool;
   Hbit_Otwórz_Z2 AT %M12.4 : Bool;
   CMD_Open_Z_2 AT %M54.5 : Bool;   // załącz otwieranie
   inputAumaawariaZ_2 AT %M54.1 : Bool;   // znacznik wejście
   Hbit_REN_Z2 AT %M12.2 : Bool;
   isAUMA_Z_2 AT %M44.0 : Bool;   // przęłącznik wymiany na AUMA
   inputAumaautomatZ_2 AT %M53.7 : Bool;   // znacznik wejście
   setAlarm_Moment_Z_2 AT %M54.4 : Bool;   // znacznik alarmu od momentówki w trybie zdalnym (aut/mamnual)
   setSVMO_Z_2 AT %M54.2 : Bool;   // Znacznik polecenia otwórz w trybie automat
   isGotowość_Z_2 AT %M53.0 : Bool;   // bit gotowości wspólny
   inputOtwartaZ_2 AT %M53.2 : Bool;   // znacznik wejście
   CMD_Awaria_Z_2 AT %M54.7 : Bool;   // Awaria zbiorcza
   CMD_Close_Z_2 AT %M54.6 : Bool;   // załącz zamykanie
   inputAumagotowośćZ_2 AT %M54.0 : Bool;   // znacznik wejście
   edge_Hz_Z2 AT %M92.0 : Bool;   // pamięć zbocza 1 Hz
END_VAR

VAR_GLOBAL   // PLC tag table "Z3"
   Hbit_Alarm_Z3 AT %M14.0 : Bool;
   CMD_Open_Z_3 AT %M57.5 : Bool;   // załącz otwieranie
   Hbit_Reset_Z3 AT %M14.6 : Bool;
   CMD_Awaria_Z_3 AT %M57.7 : Bool;   // Awaria zbiorcza
   inputOtwartaZ_3 AT %M56.2 : Bool;   // znacznik wejście
   setAlarm_Moment_Z_3 AT %M57.4 : Bool;   // znacznik alarmu od momentówki w trybie zdalnym (aut/mamnual)
   inputRuch_Z_3 AT %M56.4 : Bool;
   setSVMO_Z_3 AT %M57.2 : Bool;   // Znacznik polecenia otwórz w trybie automat
   CMD_Close_Z_3 AT %M57.6 : Bool;   // załącz zamykanie
   Byte_Status_Z3 AT %MW14 : Word;   // Słowo statusu napędu
   isAUMA_Z_3 AT %M52.4 : Bool;   // przęłącznik wymiany na AUMA
   inputAumagotowośćZ_3 AT %M57.0 : Bool;   // znacznik wejście
   Hbit_Auto_Manu_Z3 AT %M14.7 : Bool;
   inputAumalokalneZ_3 AT %M56.6 : Bool;   // znacznik wejście
   Hbit_Zamknieta_Z3 AT %M14.3 : Bool;
   setSVMC_Z_3 AT %M57.3 : Bool;   // Znacznik polecenia zamknij w trybie automat
   Hbit_REN_Z3 AT %M14.2 : Bool;
   Hbit_Otwórz_Z3 AT %M14.4 : Bool;
   inputAumaawariaZ_3 AT %M57.1 : Bool;   // znacznik wejście
   inputAumaautomatZ_3 AT %M56.7 : Bool;   // znacznik wejście
   inputREMT_Z_3 AT %M56.1 : Bool;   // znacznik wejście zdalne
   inputAwariaMomentZ_3 AT %M56.5 : Bool;   // znacznik wejście
   isGotowość_Z_3 AT %M56.0 : Bool;   // bit gotowości wspólny
   Hbit_Otwarta_Z3 AT %M14.1 : Bool;
   inputZamkniętaZ_3 AT %M56.3 : Bool;   // znacznik wejście
   Hbit_Zamknij_Z3 AT %M14.5 : Bool;
END_VAR

VAR_GLOBAL   // PLC tag table "Z4"
   Hbit_Auto_Manu_Z4 AT %M16.7 : Bool;
   Hbit_Otwarta_Z4 AT %M16.1 : Bool;
   inputAumagotowośćZ_4 AT %M60.0 : Bool;   // znacznik wejście
   CMD_Awaria_Z_4 AT %M60.7 : Bool;   // Awaria zbiorcza
   setSVMO_Z_4 AT %M60.2 : Bool;   // Znacznik polecenia otwórz w trybie automat
   Hbit_Reset_Z4 AT %M16.6 : Bool;
   inputAumalokalneZ_4 AT %M59.6 : Bool;   // znacznik wejście
   Hbit_Alarm_Z4 AT %M16.0 : Bool;
   inputRuch_Z_4 AT %M59.4 : Bool;
   inputAwariaMomentZ_4 AT %M59.5 : Bool;   // znacznik wejście
   Hbit_Otwórz_Z4 AT %M16.4 : Bool;
   inputAumaautomatZ_4 AT %M59.7 : Bool;   // znacznik wejście
   Hbit_REN_Z4 AT %M16.2 : Bool;
   setAlarm_Moment_Z_4 AT %M60.4 : Bool;   // znacznik alarmu od momentówki w trybie zdalnym (aut/mamnual)
   isGotowość_Z_4 AT %M59.0 : Bool;   // bit gotowości wspólny
   isAUMA_Z_4 AT %M52.5 : Bool;   // przęłącznik wymiany na AUMA
   Hbit_Zamknieta_Z4 AT %M16.3 : Bool;
   inputREMT_Z_4 AT %M59.1 : Bool;   // znacznik wejście zdalne
   Hbit_Zamknij_Z4 AT %M16.5 : Bool;
   inputAumaawariaZ_4 AT %M60.1 : Bool;   // znacznik wejście
   inputOtwartaZ_4 AT %M59.2 : Bool;   // znacznik wejście
   Byte_Status_Z4 AT %MW16 : Word;   // Słowo statusu napędu
   inputZamkniętaZ_4 AT %M59.3 : Bool;   // znacznik wejście
   setSVMC_Z_4 AT %M60.3 : Bool;   // Znacznik polecenia zamknij w trybie automat
   CMD_Close_Z_4 AT %M60.6 : Bool;   // załącz zamykanie
   CMD_Open_Z_4 AT %M60.5 : Bool;   // załącz otwieranie
   edge_Hz_Z4 AT %M92.1 : Bool;   // pamięć zbocza 1 Hz
END_VAR

VAR_GLOBAL   // PLC tag table "Z5"
   inputAwariaMomentZ_5 AT %M62.5 : Bool;   // znacznik wejście
   inputRuch_Z_5 AT %M62.4 : Bool;
   inputAumalokalneZ_5 AT %M62.6 : Bool;   // znacznik wejście
   Hbit_Zamknij_Z5 AT %M18.5 : Bool;
   inputOtwartaZ_5 AT %M62.2 : Bool;   // znacznik wejście
   Hbit_Otwarta_Z5 AT %M18.1 : Bool;
   setSVMC_Z_5 AT %M63.3 : Bool;   // Znacznik polecenia zamknij w trybie automat
   CMD_Close_Z_5 AT %M63.6 : Bool;   // załącz zamykanie
   inputAumaautomatZ_5 AT %M62.7 : Bool;   // znacznik wejście
   Hbit_Auto_Manu_Z5 AT %M18.7 : Bool;
   CMD_Open_Z_5 AT %M63.5 : Bool;   // załącz otwieranie
   inputAumagotowośćZ_5 AT %M63.0 : Bool;   // znacznik wejście
   CMD_Awaria_Z_5 AT %M63.7 : Bool;   // Awaria zbiorcza
   setSVMO_Z_5 AT %M63.2 : Bool;   // Znacznik polecenia otwórz w trybie automat
   Hbit_Zamknieta_Z5 AT %M18.3 : Bool;
   Hbit_Alarm_Z5 AT %M18.0 : Bool;
   isAUMA_Z_5 AT %M52.6 : Bool;   // przęłącznik wymiany na AUMA
   inputAumaawariaZ_5 AT %M63.1 : Bool;   // znacznik wejście
   Hbit_Reset_Z5 AT %M18.6 : Bool;
   isGotowość_Z_5 AT %M62.0 : Bool;   // bit gotowości wspólny
   Byte_Status_Z5 AT %MW18 : Word;   // Słowo statusu napędu
   Hbit_REN_Z5 AT %M18.2 : Bool;
   inputREMT_Z_5 AT %M62.1 : Bool;   // znacznik wejście zdalne
   inputZamkniętaZ_5 AT %M62.3 : Bool;   // znacznik wejście
   setAlarm_Moment_Z_5 AT %M63.4 : Bool;   // znacznik alarmu od momentówki w trybie zdalnym (aut/mamnual)
   Hbit_Otwórz_Z5 AT %M18.4 : Bool;
END_VAR

VAR_GLOBAL   // PLC tag table "Z6"
   inputAumagotowośćZ_6 AT %M65.0 : Bool;   // znacznik wejście
   Hbit_Reset_Z6 AT %M20.6 : Bool;
   Hbit_Zamknij_Z6 AT %M20.5 : Bool;
   inputAumaautomatZ_6 AT %M64.7 : Bool;   // znacznik wejście
   setSVMO_Z_6 AT %M65.2 : Bool;   // Znacznik polecenia otwórz w trybie automat
   inputAumalokalneZ_6 AT %M64.6 : Bool;   // znacznik wejście
   Hbit_Auto_Manu_Z6 AT %M20.7 : Bool;
   inputREMT_Z_6 AT %M64.1 : Bool;   // znacznik wejście zdalne
   inputAwariaMomentZ_6 AT %M64.5 : Bool;   // znacznik wejście
   Hbit_Otwórz_Z6 AT %M20.4 : Bool;
   isAUMA_Z_6 AT %M52.7 : Bool;   // przęłącznik wymiany na AUMA
   Hbit_REN_Z6 AT %M20.2 : Bool;
   CMD_Open_Z_6 AT %M65.5 : Bool;   // załącz otwieranie
   Hbit_Alarm_Z6 AT %M20.0 : Bool;
   Hbit_Otwarta_Z6 AT %M20.1 : Bool;
   CMD_Awaria_Z_6 AT %M65.7 : Bool;   // Awaria zbiorcza
   Hbit_Zamknieta_Z6 AT %M20.3 : Bool;
   CMD_Close_Z_6 AT %M65.6 : Bool;   // załącz zamykanie
   inputRuch_Z_6 AT %M64.4 : Bool;
   setSVMC_Z_6 AT %M65.3 : Bool;   // Znacznik polecenia zamknij w trybie automat
   isGotowość_Z_6 AT %M64.0 : Bool;   // bit gotowości wspólny
   Byte_Status_Z6 AT %MW20 : Word;   // Słowo statusu napędu
   setAlarm_Moment_Z_6 AT %M65.4 : Bool;   // znacznik alarmu od momentówki w trybie zdalnym (aut/mamnual)
   inputZamkniętaZ_6 AT %M64.3 : Bool;   // znacznik wejście
   inputOtwartaZ_6 AT %M64.2 : Bool;   // znacznik wejście
   inputAumaawariaZ_6 AT %M65.1 : Bool;   // znacznik wejście
   edge_Hz_Z6 AT %M92.2 : Bool;   // pamięć zbocza 1 Hz
END_VAR

VAR_GLOBAL   // PLC tag table "Z7"
   inputAumagotowośćZ_7 AT %M67.0 : Bool;   // znacznik wejście
   Hbit_Otwórz_Z7 AT %M22.4 : Bool;
   inputAwariaMomentZ_7 AT %M66.5 : Bool;   // znacznik wejście
   setAlarm_Moment_Z_7 AT %M67.4 : Bool;   // znacznik alarmu od momentówki w trybie zdalnym (aut/mamnual)
   isAUMA_Z_7 AT %M44.1 : Bool;   // przęłącznik wymiany na AUMA
   Hbit_Zamknieta_Z7 AT %M22.3 : Bool;
   Byte_Status_Z7 AT %MW22 : Word;   // Słowo statusu napędu
   CMD_Open_Z_7 AT %M67.5 : Bool;   // załącz otwieranie
   inputOtwartaZ_7 AT %M66.2 : Bool;   // znacznik wejście
   inputREMT_Z_7 AT %M66.1 : Bool;   // znacznik wejście zdalne
   inputAumaautomatZ_7 AT %M66.7 : Bool;   // znacznik wejście
   Hbit_Alarm_Z7 AT %M22.0 : Bool;
   CMD_Close_Z_7 AT %M67.6 : Bool;   // załącz zamykanie
   inputRuch_Z_7 AT %M66.4 : Bool;
   setSVMC_Z_7 AT %M67.3 : Bool;   // Znacznik polecenia zamknij w trybie automat
   setSVMO_Z_7 AT %M67.2 : Bool;   // Znacznik polecenia otwórz w trybie automat
   Hbit_Auto_Manu_Z7 AT %M22.7 : Bool;
   inputAumaawariaZ_7 AT %M67.1 : Bool;   // znacznik wejście
   CMD_Awaria_Z_7 AT %M67.7 : Bool;   // Awaria zbiorcza
   inputAumalokalneZ_7 AT %M66.6 : Bool;   // znacznik wejście
   Hbit_Reset_Z7 AT %M22.6 : Bool;
   isGotowość_Z_7 AT %M66.0 : Bool;   // bit gotowości wspólny
   Hbit_Otwarta_Z7 AT %M22.1 : Bool;
   Hbit_Zamknij_Z7 AT %M22.5 : Bool;
   inputZamkniętaZ_7 AT %M66.3 : Bool;   // znacznik wejście
   Hbit_REN_Z7 AT %M22.2 : Bool;
END_VAR

VAR_GLOBAL   // PLC tag table "Z8"
   inputAumagotowośćZ_8 AT %M69.0 : Bool;   // znacznik wejście
   setAlarm_Moment_Z_8 AT %M69.4 : Bool;   // znacznik alarmu od momentówki w trybie zdalnym (aut/mamnual)
   CMD_Awaria_Z_8 AT %M69.7 : Bool;   // Awaria zbiorcza
   isGotowość_Z_8 AT %M68.0 : Bool;   // bit gotowości wspólny
   inputAwariaMomentZ_8 AT %M68.5 : Bool;   // znacznik wejście
   inputOtwartaZ_8 AT %M68.2 : Bool;   // znacznik wejście
   Hbit_Reset_Z8 AT %M24.6 : Bool;
   setSVMO_Z_8 AT %M69.2 : Bool;   // Znacznik polecenia otwórz w trybie automat
   inputRuch_Z_8 AT %M68.4 : Bool;
   Hbit_Otwórz_Z8 AT %M24.4 : Bool;
   CMD_Close_Z_8 AT %M69.6 : Bool;   // załącz zamykanie
   inputAumaawariaZ_8 AT %M69.1 : Bool;   // znacznik wejście
   setSVMC_Z_8 AT %M69.3 : Bool;   // Znacznik polecenia zamknij w trybie automat
   Hbit_Alarm_Z8 AT %M24.0 : Bool;
   Hbit_Zamknij_Z8 AT %M24.5 : Bool;
   CMD_Open_Z_8 AT %M69.5 : Bool;   // załącz otwieranie
   inputZamkniętaZ_8 AT %M68.3 : Bool;   // znacznik wejście
   Hbit_Zamknieta_Z8 AT %M24.3 : Bool;
   inputREMT_Z_8 AT %M68.1 : Bool;   // znacznik wejście zdalne
   Hbit_REN_Z8 AT %M24.2 : Bool;
   isAUMA_Z_8 AT %M44.2 : Bool;   // przęłącznik wymiany na AUMA
   inputAumalokalneZ_8 AT %M68.6 : Bool;   // znacznik wejście
   Hbit_Otwarta_Z8 AT %M24.1 : Bool;
   Hbit_Auto_Manu_Z8 AT %M24.7 : Bool;
   Byte_Status_Z8 AT %MW24 : Word;   // Słowo statusu napędu
   inputAumaautomatZ_8 AT %M68.7 : Bool;   // znacznik wejście
   edge_Hz_Z8 AT %M92.3 : Bool;   // pamięć zbocza 1 Hz
END_VAR

VAR_GLOBAL   // PLC tag table "Z9"
   isGotowość_Z_9 AT %M70.0 : Bool;   // bit gotowości wspólny
   inputAumaawariaZ_9 AT %M71.1 : Bool;   // znacznik wejście
   Hbit_REN_Z9 AT %M26.2 : Bool;
   CMD_Close_Z_9 AT %M71.6 : Bool;   // załącz zamykanie
   inputZamkniętaZ_9 AT %M70.3 : Bool;   // znacznik wejście
   inputAumaautomatZ_9 AT %M70.7 : Bool;   // znacznik wejście
   inputAumagotowośćZ_9 AT %M71.0 : Bool;   // znacznik wejście
   Hbit_Otwórz_Z9 AT %M26.4 : Bool;
   setAlarm_Moment_Z_9 AT %M71.4 : Bool;   // znacznik alarmu od momentówki w trybie zdalnym (aut/mamnual)
   Hbit_Reset_Z9 AT %M26.6 : Bool;
   Hbit_Zamknieta_Z9 AT %M26.3 : Bool;
   Hbit_Auto_Manu_Z9 AT %M26.7 : Bool;
   Byte_Status_Z9 AT %MW26 : Word;   // Słowo statusu napędu
   inputAwariaMomentZ_9 AT %M70.5 : Bool;   // znacznik wejście
   CMD_Awaria_Z_9 AT %M71.7 : Bool;   // Awaria zbiorcza
   CMD_Open_Z_9 AT %M71.5 : Bool;   // załącz otwieranie
   Hbit_Zamknij_Z9 AT %M26.5 : Bool;
   isAUMA_Z_9 AT %M52.1 : Bool;   // przęłącznik wymiany na AUMA
   Hbit_Alarm_Z9 AT %M26.0 : Bool;
   inputOtwartaZ_9 AT %M70.2 : Bool;   // znacznik wejście
   setSVMC_Z_9 AT %M71.3 : Bool;   // Znacznik polecenia zamknij w trybie automat
   inputRuch_Z_9 AT %M70.4 : Bool;
   Hbit_Otwarta_Z9 AT %M26.1 : Bool;
   inputREMT_Z_9 AT %M70.1 : Bool;   // znacznik wejście zdalne
   inputAumalokalneZ_9 AT %M70.6 : Bool;   // znacznik wejście
   setSVMO_Z_9 AT %M71.2 : Bool;   // Znacznik polecenia otwórz w trybie automat
END_VAR

VAR_GLOBAL   // PLC tag table "Zasuwy"
   isAutPumping AT %M80.6 : Bool;   // wybrana opcja automatycznego sterowania pompowanie lub dosilanie
   isPumping AT %M80.4 : Bool;   // wybrana opcja przepompowywanie na miasto
   isTime_FillingOn AT %M90.4 : Bool;   // znacznik start napełnianie
   isTime_FillingOff AT %M90.5 : Bool;   // znacznik stop napełnianie
   isTime_EptyingOn AT %M90.6 : Bool;   // znacznik start przetłaczanie
   isRecharging AT %M80.5 : Bool;   // wybrana opcja dosilania na magistralę
   isTime_EptyingOff AT %M90.7 : Bool;   // znacznik stop przetłaczanie
   inputREM_Zasuwy AT %M50.4 : Bool;   // znacznik wejście zdalane
   isManual AT %M81.1 : Bool;   // tryb sterowania manualny
   memTriggerClose_setValue_Z11 AT %M90.1 : Bool;   // pamięć zbocza przekazania nowego meldunku dla otwierania
   memTriggerOpen_setValue_Z10 AT %M90.0 : Bool;   // pamięć zbocza przekazania nowego meldunku
END_VAR

VAR_GLOBAL   // PLC tag table "zbiorniki"
   set_HWork_Tank_3 AT %M45.2 : Bool;   // bit statusu aktywacji zbiornika do pracy w trybie sekwencji
   set_HWork_Tank_1 AT %M45.0 : Bool;   // bit statusu aktywacji zbiornika do pracy w trybie sekwencji
   set_HWork_Tank_2 AT %M45.1 : Bool;   // bit statusu aktywacji zbiornika do pracy w trybie sekwencji
   set_HWork_Tank_4 AT %M45.3 : Bool;   // bit statusu aktywacji zbiornika do pracy w trybie sekwencji
   mem_set_auto_zb_3 AT %M82.2 : Bool;   // ustawione w sekwencji jako aktywna
   blok_tank_3 AT %M82.6 : Bool;   // jest zablokowany po pracy w sekwencji
   blok_tank_1 AT %M82.4 : Bool;   // jest zablokowany po pracy w sekwencji
   mem_set_auto_zb_2 AT %M82.1 : Bool;   // ustawione w sekwencji jako aktywna
   blok_tank_4 AT %M82.7 : Bool;   // jest zablokowany po pracy w sekwencji
   act_Eptying AT %M45.4 : Bool;   // trwa procedura pompowania
   mem_set_auto_zb_1 AT %M82.0 : Bool;   // ustawione w sekwencji jako aktywna
   memTrig_set_manual_zb_4 AT %M83.3 : Bool;   // ustaw w automat zasuwę aktywnego zbiornika
   memTrig_set_manual_zb_3 AT %M83.2 : Bool;   // ustaw w automat zasuwę aktywnego zbiornika
   memTrig_set_manual_zb_1 AT %M83.0 : Bool;   // ustaw w automat zasuwę aktywnego zbiornika
   blok_tank_2 AT %M82.5 : Bool;   // jest zablokowany po pracy w sekwencji
   act_Filling AT %M45.5 : Bool;   // trwa procedura napełniania
   mem_set_auto_zb_4 AT %M82.3 : Bool;   // ustawione w sekwencji jako aktywna
   memTrig_set_manual_zb_2 AT %M83.1 : Bool;   // ustaw w automat zasuwę aktywnego zbiornika
END_VAR

TYPE "stt_OB82"
// stored: IsFailsafeCompliant false
   STRUCT
      ErrorTimestamp : DTL;   // //time error occurs
      IO_State : Word;   // //Contains the I/O status of the diagnostics-capable module.
      LADDR : HW_ANY;   // //HW-ID
      Channel : UInt;   // //Channel number
      MultiError : Bool;   // //= 1, if there is more than one error
   END_STRUCT;
END_TYPE

TYPE "typeMbClient"
// stored: IsFailsafeCompliant false
   STRUCT
      req : Bool;   // Activates the requested transmission if TRUE
      disconnect : Bool;   // Initiates a disconnect operation
      mode : USInt;   // Specifies the type of request: read, write or diagnostic
      mbDataAddr : UDInt := 40066;   // Specifies the starting address of the data to be accessed in the Modbus client
      connect { S7_SetPoint := 'True'} : TCON_IP_v4;   // Reference to the connection parameters
   END_STRUCT;
   // connect.InterfaceId := 64;
   // connect.ID := 1;
   // connect.ActiveEstablished := true;
   // connect.RemoteAddress.ADDR[1] := 192;
   // connect.RemoteAddress.ADDR[2] := 168;
   // connect.RemoteAddress.ADDR[3] := 0;
   // connect.RemotePort := 502;
END_TYPE

TYPE "typVARIANT"
// stored: IsFailsafeCompliant false
   STRUCT
      VARIANT : Array[0..1] of Bool;
   END_STRUCT;
END_TYPE

TYPE "typeDataInverter_Byte"
// stored: IsFailsafeCompliant false
   STRUCT
      typeDataInverter_byte : Array[0..0] of Byte;   // Typ dane byte, falownik
   END_STRUCT;
END_TYPE

TYPE "typeDataInverter_DWord"
// stored: IsFailsafeCompliant false
   STRUCT
      typeDataInverter_Dword : Array[0..0] of DInt;   // dane dword, falownik
   END_STRUCT;
END_TYPE

TYPE "typeDataInverter_Real"
// stored: IsFailsafeCompliant false
   STRUCT
      typeDataInverter_real : Array[0..0] of Real;   // dane real, falownik
   END_STRUCT;
END_TYPE

TYPE "typeDataInverter_Word"
// stored: IsFailsafeCompliant false
   STRUCT
      typeDataInverter_int : Array[0..0] of Int;   // Typ danej Int, falownik
   END_STRUCT;
END_TYPE

TYPE "typeDataMPP04_Int"
// stored: IsFailsafeCompliant false
   STRUCT
      data : Array[0..1] of Int;
   END_STRUCT;
END_TYPE

TYPE "typeDataMPP04_int_1"
// stored: IsFailsafeCompliant false
   STRUCT
      data : Array[0..0] of Int;
   END_STRUCT;
END_TYPE

TYPE "typeDataMPP04_real"
// stored: IsFailsafeCompliant false
   STRUCT
      data : Array[0..0] of Real;
   END_STRUCT;
END_TYPE

TYPE "typeModbusCommLoad"
// stored: IsFailsafeCompliant false
   STRUCT
      done : Bool := FALSE;   // Boolean indicating completion without error
      error : Bool := FALSE;   // Boolean indicating completion with error
      status : Word := W#16#0;   // Status or error code of the completed operation
      errorStatus : Word := W#16#0;   // Error code of the faulty operation
   END_STRUCT;
END_TYPE

TYPE "typeModbusMaster"
// stored: IsFailsafeCompliant false
   STRUCT
      req : Bool := FALSE;   // The enable to initiate a Modbus master request
      mbAddr : UInt;   // The station address of the Modbus slave
      mode : USInt := 0;   // Specifies a read, write, or diagnostic operation
      dataAddr : UDInt := 0;   // The Modbus data address
      dataLen : UInt := 0;   // The Modbus data length
      done : Bool := FALSE;   // Boolean indicating completion without error
      busy : Bool := FALSE;   // Boolean indicating operation in progress
      error : Bool := FALSE;   // Boolean indicating completion with error
      status : Word := W#16#0;   // Status or error code of the completed operation
      errorStatus : Word := W#16#0;   // Error code of the faulty operation
   END_STRUCT;
END_TYPE

TYPE "typeModbusSlave"
// stored: IsFailsafeCompliant false
   STRUCT
      NDR : Bool := FALSE;   // New data ready: 1: Indicates that data has been read by the Modbus master No new data
      mbAddr : UInt;   // Station address of the Modbus slave (address range: 0 to 255)
      done : Bool := FALSE;   // Boolean indicating completion without error
      dr : Bool := FALSE;   // Read data: 0: No data read1: Indicates that data has been read by the Modbus master
      error : Bool := FALSE;   // Boolean indicating completion with error
      status : Word := W#16#0;   // Status or error code of the completed operation
      errorStatus : Word := W#16#0;   // Error code of the faulty operation
   END_STRUCT;
END_TYPE

DATA_BLOCK "DB31_HMI_AreaPointer"   // DB31
{ S7_Optimized_Access := 'FALSE' }
VERSION : 0.1
// stored: AutoNumber false, DBAccessibleFromOPCUA true, IsOnlyStoredInLoadMemory false, IsWriteProtectedInAS false
   VAR
      Coordination : Word;
      DateTime : DTL;
      JobMailbox : Array[0..3] of Word;
      DataRecord : Array[0..4] of Word;
      ProjectID : Word;
      ScreenNumber : Array[0..4] of Word;
      DateTimePLC : Struct
         DateTime : DTL;
         Reserve_01 : Word;
         Reserve_02 : Word;
      END_STRUCT;
      getPLCMode : Int;
      retValueTime : Word;
      cpuSatus : Bool;   // bit satus CPU (0-RUN, 1-RESATR)
   END_VAR
BEGIN
END_DATA_BLOCK

DATA_BLOCK "Dane_ComunicationControlHMI"   // DB29
TITLE = WatchDog HMI-Krata - S7-Krata
{ S7_Optimized_Access := 'FALSE' }
AUTHOR : rtecmer
VERSION : 0.1
// stored: AutoNumber true, DBAccessibleFromOPCUA true, IsOnlyStoredInLoadMemory false, IsWriteProtectedInAS false
   VAR
      Data_czas_loc : DTL;   // Zegar dla panelu HMI Krata
      WatchDog_WinCC : Word;   // Zmienna kordynująca kontrolę komunikacji od strony PC WinCC.
      "CoordinationPLC-PLC" : Int;   // Kontrola komunikacji z PLC-PLC
      Data_czas_sys : DTL;   // Zegar dla panelu HMI Krata
      Data_czasHMI : DTL;   // Zegar czytany z funkcji RTC (FC44) zapas
      tempCoordinationHMIRS5 : Int;   // Kontrola CoorditionHMI KDN
      tempWatchDog_WinCC : Word;   // Zmienna kordynująca kontrolę komunikacji od strony PC WinCC.
   END_VAR
BEGIN
END_DATA_BLOCK

DATA_BLOCK "Data_Czas_synch"   // DB32
{ S7_Optimized_Access := 'FALSE' }
VERSION : 0.1
// stored: AutoNumber false, DBAccessibleFromOPCUA true, IsOnlyStoredInLoadMemory false, IsWriteProtectedInAS false
   VAR
      Time_Local_read : DTL;
      Time_System_read : DTL;
      Time_System_write : DTL;
      zegar : Time_Of_Day;
      memTrig_Week : Bool;   // pamieć zbocza uruchomienia funkcji tygodniowej
      memTrigRes_Week : Bool;   // pamieć zbocza resetu odmierzonej doby
   END_VAR
BEGIN
END_DATA_BLOCK

DATA_BLOCK "DB10_instance_SCADA"   // DB10
TITLE = SCADA
{ S7_Optimized_Access := 'FALSE' }
AUTHOR : rtecmer
VERSION : 0.1
// stored: AutoNumber false, DBAccessibleFromOPCUA true, IsOnlyStoredInLoadMemory false, IsWriteProtectedInAS false
   VAR
      Clock : Time;
      Watchdog : Int;
      instZ1 : Word := 33924;   // status zasuwy
      instZ2 : Word := 33924;   // status zasuwy
      instZ3 : Word := 33924;   // status zasuwy
      instZ4 : Word := 33924;   // status zasuwy
      instZ5 : Word := 33924;   // status zasuwy
      instZ6 : Word := 33924;   // status zasuwy
      instZ7 : Word := 33924;   // status zasuwy
      instZ8 : Word := 33924;   // status zasuwy
      instZ9 : Word := 33924;   // status zasuwy
      instZ10 : Word := 33924;   // status zasuwy
      actPoziomZbiornik_1 : Real;   // aktualny poziom w zbirniku
      actPoziomZbiornik_2 : Real := 0.0;   // aktualny poziom w zbirniku
      actPoziomZbiornik_3 : Real := 0.0;   // aktualny poziom w zbirniku
      actPoziomZbiornik_4 : Real := 0.0;   // aktualny poziom w zbirniku
      actPoziomZbiornik_5 : Real := 0.0;   // aktualny poziom w zbirniku
      actPrzepływ_Q2 : Real;   // aktualny przepływ Q2 - studnia pomiarowa przed pompownią
      sumPrzepływVF_Q2 : Real;   // suma przepływu
      statusPrzepływVR_Q2 : Real := 0.0;   // status przepływomierza
      setPołożenieZ10 : Word := 40;   // zadany [%] otwarcia
      actPołożenieZ10 : Word;   // aktualny [%] otwarcia
      rtu_mpp04_2error_status : Word;   // status błędu modbus przepływomierz Q2
      ModelSterowania : Word;   // Sygnały sterowania strategią pompownia - 0= wyłaczone, 1=dosilanie, 2=przetłaczanie,3=automat, 4=ręczne
      TrybSterowania : Word;   // Tryb 0-wyłączony, 1- Dobowy, 2- Tygodniowy, 3-Ręczny
      "Alarms only" : Word;   // Instancja alarmów (bit 68.0 - Error komunikacji z HMI)
      setPoziomNapełniania : Real := 550.0;   // zadana wartość napełniania
      setPoziomOpróżnianai : Real := 30.0;   // zadana wartość opróżniania
      "actCiśnienie-magistralaB5" : Real := 6.6;   // ciśnienie na przewodzie zasilania 9magistrala)
      rtu_step_reset : Bool;   // reset modbus RTU
      actTime_FillingOn : Real;   // godzina start napełnianie
      actTime_FillingOff : Real;   // godzina stop napełnianie
      actTime_EptyingOn : Real;   // godzina start przetłaczanie
      actTime_EptyingOff : Real;   // godzina stop przetłaczanie
      actTime : Real;   // czas aktualny
      actDTL_FillingOn : DTL := DTL#2022-08-02-00:05:00;   // zmienna DTL napełnianie start
      actDTL_FillingOff : DTL := DTL#2022-08-02-17:00:00.000000003;   // zmienna DTL napełnianie stop
      actDTL_pumpingOn : DTL := DTL#2022-08-02-18:00:00.000000003;   // zmienna DTL przetłaczanie start
      actDTL_pumpingOff : DTL := DTL#2022-08-02-23:59:00.000000001;   // zmienna DTL przetłaczanie stop
      actDTL_RechargingOn : DTL := DTL#2022-08-02-18:00:00.000000013;   // zmienna DTL dosilanie start
      actDTL_RechargingOff : DTL := DTL#2022-08-02-23:59:00.000000003;   // zmienna DTL dosilanie stop
      reset_modbus_TCP : Bool;   // reset modbus TCP
      instConrol_ManAut_1 : Int := 0;   // Bity przełączenia trybu pracy napędów / 40019 Bity przełączenia trybu pracy napędów M1-M4, Zasuwami Z1, Z2, Z3, Z4
      instConrol_ManAut_2 : Int := 0;   // Bity przełączenia trybu pracy napędów / 40020 Bity przełączenia trybu pracy napędów Z5, Z6, Z7, Z8, Z9, Z10, Z11, Z12
   END_VAR
BEGIN
END_DATA_BLOCK

DATA_BLOCK "Parametryzacja"   // DB12
TITLE = Konfiguracja parametrów
{ S7_Optimized_Access := 'FALSE' }
AUTHOR : rtecmer
VERSION : 0.1
// Dane konfiguracji parametrów przepływomierza, sond pomiarowych, przetworników
// stored: AutoNumber true, DBAccessibleFromOPCUA true, IsOnlyStoredInLoadMemory false, IsWriteProtectedInAS false
   VAR RETAIN
      "Setting analog" : Struct   // Parametry przetworników analogowych
         maxPrzepływomierz_Q2 : Real := 600.0;   // nastawa konfiguracji przetwornika przepływomierza wartość max przepływ
         minPrzepływomierz_Q2 : Real := 0.0;   // nastawa konfiguracji przetwornika przepływomierza wartość min przepływ
         maxPrzetwornikCiśnienia_B5 : Real := 16.0;   // nastawa konfiguracji przetwornika
         minPrzetwornikCiśnienia_B5 : Real := 0.0;   // nastawa konfiguracji przetwornika
         maxSondaHydro : Real := 1000.0;   // nastawa konfiguracji przetwornika
         minSondaHydro : Real := 0.0;   // nastawa konfiguracji przetwornika
      END_STRUCT;
      "Setting Controll" : Struct   // Parametry nastaw w procesie sterowania
         alarmMin_CiśnienieGranica : Real := 6.5;   // minimalne dopuszczalne ciśnienie Granica
         alarmMax_CiśnienieGranica : Real := 10.0;   // minimalne dopuszczalne ciśnienie Granica
         maxZbiorniki : Real := 600.0;   // stan alarmowy poziomu
         minZbiorniki : Real := 100.0;   // stan alarmowy poziomu
         max_położenie_Z10 : Real := 101.0;   // stan alarmowy położenia
         min_położenie_Z10 : Real := -0.5;   // stan alarmowy położenia
         setPoziomNapełniania : Real := 550.0;   // zadana wartość napełniania
         setPoziomOpróżnianai : Real := 30.0;   // zadana wartość opróżniania
         setPołożenieZ10 : Word;   // zadany [%] otwarcia
         tmpPołożenieZ10 : Word;   // tymczasowa zadany [%] otwarcia do przekazania
         ModelSterowania : Word;   // Zmienna przyjmująca wartość dziesiętnią oznaczającą model sterowania
         TrybSterowania : Word;   // Tryb 0-wyłączony, 1- Dobowy, 2- Tygodniowy, 3-Ręczny
      END_STRUCT;
      "Status drivers" : Struct   // Status napedów
         instZ1 : Word;   // status zasuwy
         instZ2 : Word;   // status zasuwy
         instZ3 : Word;   // status zasuwy
         instZ4 : Word;   // status zasuwy
         instZ5 : Word;   // status zasuwy
         instZ6 : Word;   // status zasuwy
         instZ7 : Word;   // status zasuwy
         instZ8 : Word;   // status zasuwy
         instZ9 : Word;   // status zasuwy
         instZ10 : Word;   // status zasuwy
      END_STRUCT;
      "Controls Tanks" : Struct   // Sterowanie zbiornikami
         aktywny_Zbiornik_1 : Bool;   // zbiornik włączony w cykl pracy 1=aktywny
         aktywny_Zbiornik_2 : Bool;   // zbiornik włączony w cykl pracy 1=aktywny
         aktywny_Zbiornik_3 : Bool;   // zbiornik włączony w cykl pracy 1=aktywny
         aktywny_Zbiornik_4 : Bool;   // zbiornik włączony w cykl pracy 1=aktywny
         aktywne_Napełnianie : Bool;   // bit aktywacji funkcji napełniania
         "aktywne _Przetłaczanie" : Bool;   // bit aktywacji funkcji przetłaczania
         aktywne_Dosilanie : Bool;   // bit aktywacji funkcji dosilania
      END_STRUCT;
      "Time Tanks" : Struct
         Start_napełnianie : DTL := DTL#1970-01-01-23:55:00;
         Stop_napełnianie : DTL := DTL#1970-01-01-16:00:00;
         Start_przetłaczanie_1 : DTL := DTL#1970-01-01-18:00:00;
         Stop_przetłaczanie_1 : DTL := DTL#1970-01-01-23:40:00;
         Start_dosilanie_1 : DTL := DTL#1970-01-01-18:00:00;
         Stop_dosilanie_1 : DTL := DTL#1970-01-01-23:40:00;
         Tank_bocking : Struct   // bity blokowania zbiornika w trybie sekwencyjnym
            blocing_tank1 : Bool;
            blocing_tank2 : Bool := false;
            blocing_tank3 : Bool := false;
            blocing_tank4 : Bool := false;
         END_STRUCT;
      END_STRUCT;
   END_VAR
BEGIN
END_DATA_BLOCK

DATA_BLOCK "Zmienne_sterujące_zbiorników"   // DB44
{ S7_Optimized_Access := 'FALSE' }
VERSION : 0.1
// stored: AutoNumber true, DBAccessibleFromOPCUA true, IsOnlyStoredInLoadMemory false, IsWriteProtectedInAS false
   VAR
      Zbiornik_1 : Struct
         active_Zb : Bool;   // znacznik aktywnego zbiornika 1= aktywny
         memRisingLevel_min_Zb : Bool;   // pamięc zbocza osiągniecia poziomu minimum w zbiorniku
         memRisingLevel_max_Zb : Bool;   // pamięc zbocza osiągniecia poziomu max w zbiorniku
         isLevelMax_Zb : Bool;   // bit osiągnieia poziomu max w zbiorniku
         isLevelMin_Zb : Bool;   // bit osiągnieia poziomu min w zbiorniku
         isFilling_Zb : Bool;   // bit aktywacji napełniania zbiornika
         isEptying_Zb { ExternalAccessible := 'False'; ExternalVisible := 'False'; ExternalWritable := 'False'} : Bool;   // bit aktywacji przetłaczania
         is_min_float_Zb : Bool;   // sygnał z pływaka minimum
         is_max_float_Zb : Bool;   // sygnał z pływaka max
         ative_Filling : Bool;   // ustawiony jako aktywny do napełniania
         active_Eptying_ : Bool;   // ustawiony jako aktywny do opróżniania
      END_STRUCT;
      Zbiornik_2 : Struct
         active_Zb : Bool;   // znacznik aktywnego zbiornika 1= aktywny
         memRisingLevel_min_Zb : Bool;   // pamięc zbocza osiągniecia poziomu minimum w zbiorniku
         memRisingLevel_max_Zb : Bool;   // pamięc zbocza osiągniecia poziomu max w zbiorniku
         isLevelMax_Zb : Bool;   // bit osiągnieia poziomu max w zbiorniku
         isLevelMin_Zb : Bool;   // bit osiągnieia poziomu min w zbiorniku
         isFilling_Zb : Bool;   // bit aktywacji napełniania zbiornika
         isEptying_Zb { ExternalAccessible := 'False'; ExternalVisible := 'False'; ExternalWritable := 'False'} : Bool;   // bit aktywacji przetłaczania
         is_min_float_Zb : Bool;   // sygnał z pływaka minimum
         is_max_float_Zb : Bool;   // sygnał z pływaka max
         ative_Filling : Bool;   // ustawiony jako aktywny do napełniania
         active_Eptying_ : Bool;   // ustawiony jako aktywny do opróżniania
      END_STRUCT;
      Zbiornik_3 : Struct
         active_Zb : Bool;   // znacznik aktywnego zbiornika 1= aktywny
         memRisingLevel_min_Zb : Bool;   // pamięc zbocza osiągniecia poziomu minimum w zbiorniku
         memRisingLevel_max_Zb : Bool;   // pamięc zbocza osiągniecia poziomu max w zbiorniku
         isLevelMax_Zb : Bool;   // bit osiągnieia poziomu max w zbiorniku
         isLevelMin_Zb : Bool;   // bit osiągnieia poziomu min w zbiorniku
         isFilling_Zb : Bool;   // bit aktywacji napełniania zbiornika
         isEptying_Zb { ExternalAccessible := 'False'; ExternalVisible := 'False'; ExternalWritable := 'False'} : Bool;   // bit aktywacji przetłaczania
         is_min_float_Zb : Bool;   // sygnał z pływaka minimum
         is_max_float_Zb : Bool;   // sygnał z pływaka max
         ative_Filling : Bool;   // ustawiony jako aktywny do napełniania
         active_Eptying_ : Bool;   // ustawiony jako aktywny do opróżniania
      END_STRUCT;
      Zbiornik_4 : Struct
         active_Zb : Bool;   // znacznik aktywnego zbiornika 1= aktywny
         memRisingLevel_min_Zb : Bool;   // pamięc zbocza osiągniecia poziomu minimum w zbiorniku
         memRisingLevel_max_Zb : Bool;   // pamięc zbocza osiągniecia poziomu max w zbiorniku
         isLevelMax_Zb : Bool;   // bit osiągnieia poziomu max w zbiorniku
         isLevelMin_Zb : Bool;   // bit osiągnieia poziomu min w zbiorniku
         isFilling_Zb : Bool;   // bit aktywacji napełniania zbiornika
         isEptying_Zb { ExternalAccessible := 'False'; ExternalVisible := 'False'; ExternalWritable := 'False'} : Bool;   // bit aktywacji przetłaczania
         is_min_float_Zb : Bool;   // sygnał z pływaka minimum
         is_max_float_Zb : Bool;   // sygnał z pływaka max
         ative_Filling : Bool;   // ustawiony jako aktywny do napełniania
         active_Eptying_ : Bool;   // ustawiony jako aktywny do opróżniania
      END_STRUCT;
      out_weekday : Bool;   // bit genetarora tygodniowego
      start_weekday : Bool;   // bit aktywacji pracy tygodniowej zbiorników
      data_sek : Word;   // licznik sekund trybu tygodniowego
      data_hour : DWord;   // licznik godzin trybu tygodniowego
      actOpenZ10 : Bool;   // bit aktywacji przekazania nowej wartości na otwarcie Z10
      actCloseZ10 : Bool;   // bit aktywacji przekazania wartości na zamknięcie [0] Z10
      testowy1 : Int;   // na potrzeby testu
   END_VAR
BEGIN
END_DATA_BLOCK

DATA_BLOCK "dbTimersForDrivers"   // DB7
{ S7_Optimized_Access := 'FALSE' }
VERSION : 0.1
// stored: AutoNumber true, DBAccessibleFromOPCUA true, IsOnlyStoredInLoadMemory false, IsWriteProtectedInAS false
   VAR
      TimerZ1 { S7_SetPoint := 'True'} : IEC_TIMER;   // Timer drivera
      TimerZ2 { S7_SetPoint := 'True'} : IEC_TIMER;   // Timer drivera
      TimerZ3 { S7_SetPoint := 'True'} : IEC_TIMER;   // Timer drivera
      TimerZ4 { S7_SetPoint := 'True'} : IEC_TIMER;   // Delay Reset Mode Work Aut
      TimerZ5 { S7_SetPoint := 'True'} : IEC_TIMER;   // Timer drivera
      TimerZ6 { S7_SetPoint := 'True'} : IEC_TIMER;   // Timer drivera
      TimerZ7 { S7_SetPoint := 'True'} : IEC_TIMER;   // Timer drivera
      TimerZ8 { S7_SetPoint := 'True'} : IEC_TIMER;   // Timer blokowania dołączenie stycznika falownika
      TimerZ9 { S7_SetPoint := 'True'} : IEC_TIMER;   // Timer blokowania dołączenie stycznika falownik
      TimerZ10 { S7_SetPoint := 'True'} : IEC_TIMER;   // Timer blokowania dołączenie stycznika falownik
      ResetBit_KasowaniaAlarm { S7_SetPoint := 'True'} : IEC_TIMER;   // Timer impulsu kasowania bitu kasowania alarmów HMI
      ispowerOK { S7_SetPoint := 'True'} : IEC_TIMER;   // Timer impulsu kasowania bitu kasowania alarmów HMI
      error_loop_modbus_tcp { S7_SetPoint := 'True'} : IEC_TIMER;   // timer kontroli obiegu petli modbus tcp
      error_loop_modbus_rtu { S7_SetPoint := 'True'} : IEC_TIMER;   // timer kontroli obiegu petli modbus rtu
      sequence_time_off : Real;   // timer kontroli zakończenie sekwencji zbiorników uaktywnia reset znacznika aktwnego zbiornika
   END_VAR
BEGIN
   TimerZ1.PT := T#30S;
   TimerZ2.PT := T#30S;
   TimerZ3.PT := T#30S;
   TimerZ4.PT := T#30S;
   TimerZ5.PT := T#30S;
   TimerZ6.PT := T#30S;
   TimerZ7.PT := T#30S;
   TimerZ8.PT := T#30S;
   TimerZ9.PT := T#30S;
   TimerZ10.PT := T#2M;
   ResetBit_KasowaniaAlarm.PT := T#2S;
   ispowerOK.PT := T#2S;
   error_loop_modbus_tcp.PT := T#45S;
   error_loop_modbus_rtu.PT := T#10S;
END_DATA_BLOCK

DATA_BLOCK "dbdane"   // DB28
{ S7_Optimized_Access := 'FALSE' }
VERSION : 0.1
// stored: AutoNumber true, DBAccessibleFromOPCUA true, IsOnlyStoredInLoadMemory false, IsWriteProtectedInAS false
   VAR RETAIN
      alarmMax_bar : Real;   // Alarmowa wartośćbar natychmiastowe wyłączenie układu
      alarmMin_bar : Int;   // pomocnicza Hz tymczasowe dla opadającego ciśnienia z Max
      Wielkość_przeływu_Q2 : Real;   // odczytana z Modbus RTU
      Licznik_objętość_VF_Q2 : Real;
      Licznik_objętość_VR_Q2 : Real;
      Licznik_różnicowy_VD_Q2 : Real;
      Stan_licz_bjętości_GF_Q2 : Real;
      Stan_licz_rózicowego_obj_GD_Q2 : Real;
      _Stan_urządzenia_Q2 : Int;
      Wielkość_przepływu_Q2_analog : Real;   // aktualny przepływ z wy analogowego
      error_step_RTu : Int;
      HourCounterP1 : DWord;   // Counter Work
      HourCounterP2 : DWord;   // Counter Work
      HourCounterP3 : DWord;   // Counter Work
      HourCounterP4 : DWord;
      Sek_P1 : Int := 1;   // Licznik sekund
      Sek_P2 : Int := 2;   // Licznik sekund
      Sek_P3 : Int := 3;   // Licznik sekund
      Sek_P4 : Int := 3;
      Edge_P1 : Bool;   // Pamięć zbocza
      Edge_P2 : Bool;   // Pamięć zbocza
      Edge_P3 : Bool;   // Pamięć zbocza
      Edge_P4 : Bool := false;
      Sek_a : Int;   // Licznik sekund
      Sek_b : Int;   // Licznik sekund
      Edge_a : Bool;   // Pamięć zbocza
      Edge_b : Bool;   // Pamięć zbocza
      Sum_sek_hur_P1 : Real := 0.01;   // Licznik sumator godzin i sekund na potrzeby wyznaczania dumchawy do pracy
      Sum_sek_hur_P2 : Real := 0.009;   // Licznik sumator godzin i sekund na potrzeby wyznaczania dumchawy do pracy
      Sum_sek_hur_P3 : Real := 0.005;   // Licznik sumator godzin i sekund na potrzeby wyznaczania dumchawy do pracy
      Sum_sek_hur_P4 : Real := 0.001;
   END_VAR
BEGIN
END_DATA_BLOCK

DATA_BLOCK "dbtags_Sterowanie"   // DB1
{ S7_Optimized_Access := 'FALSE' }
VERSION : 0.1
// stored: AutoNumber false, DBAccessibleFromOPCUA true, IsOnlyStoredInLoadMemory false, IsWriteProtectedInAS false
   VAR RETAIN
      HMI : Struct
         PhysicalUnit : String[5] := '1/min';
         Output_PWM_USInt : USInt;
         "position reached" : Bool;   // bit potwierdzenia zasuwa Z10 na pozycji
         ManualMode_visible : Bool;
         Manual_ : Bool;   // rez
         ErrorAck_1_Int : Int;
         ErrorAck_Int : Int;
         Warning_Int : Int;
         ErrorAck_Int_edge : Bool;
         ErrorAck : Bool;
         Acknowledge_visible : Bool;
         resetScreen_1 : Bool;
         resetScreen_2 : Bool := false;
         resetScreen_3 : Bool := false;
         resetScreen_4 : Bool := false;
         resetScreen_5 : Bool := false;
         resetScreen_6 : Bool := false;
         resetScreen_7 : Bool := false;
         resetScreen_8 : Bool := false;
         resetScreen_9 : Bool := false;
         resetScreen_10 : Bool := false;
         resetScreen_11 : Bool := false;
         resetScreen_12 : Bool := false;
         resetScreen_13 : Bool := false;
      END_STRUCT;
      "Z10 Pozycja" : Struct
         encoder : Word;
         rpm : Word;
      END_STRUCT;
      SetupControl : Struct
         Static_ : Bool;
      END_STRUCT;
      "Analog pomiar" : Struct
         ciśnienie_B5 : Real;
         kolman_poziom_zbiornik_1 : Real;
         kolman_poziom_zbiornik_2 : Real := 16#0;
         kolman_poziom_zbiornik_3 : Real := 16#0;
         kolman_poziom_zbiornik_4 : Real := 16#0;
         AI_ciśnienie_B5 : Real;
         AI_poziom_zbiornik_1 : Real;
         AI_poziom_zbiornik_2 : Real := 0.0;
         AI_poziom_zbiornik_3 : Real := 0.0;
         AI_poziom_zbiornik_4 : Real := 0.0;
      END_STRUCT;
   END_VAR
BEGIN
END_DATA_BLOCK

DATA_BLOCK "KALMAN_DB"   // DB45
{ S7_Optimized_Access := 'TRUE' }
VERSION : 0.1
// stored: AutoNumber false, DBAccessibleFromOPCUA true, IsOnlyStoredInLoadMemory false, IsRetainMemResEnabled false, IsWriteProtectedInAS false, MemoryReserve 250
   VAR
      kalman_P : Array[0..4] of Real;
      kalman_K : Array[0..4] of Real;
      kalman_Q : Array[0..4] of Real;
      kalman_R : Array[0..4] of Real;
      kalman_napiecie : Array[0..4] of Real;
      pomiar_napiecie : Array[0..4] of Real;
      wejscie_anal : Array[0..4] of Word;
   END_VAR
BEGIN
   // pomiar_napiecie[0] : zbiornik 1
   // pomiar_napiecie[1] : zbiornik 2
   // pomiar_napiecie[2] : zbiornik 3
   // pomiar_napiecie[3] : zbiornik 4
   // pomiar_napiecie[4] : Ciśnienie magistrala
END_DATA_BLOCK

DATA_BLOCK "EX012_ErrorBuffer_OB82"   // DB103
TITLE = BufferOB82
{ S7_Optimized_Access := 'TRUE' }
AUTHOR : Gilewski
VERSION : 0.1
// Data block for OB82 buffer
// stored: AutoNumber false, DBAccessibleFromOPCUA true, IsOnlyStoredInLoadMemory false, IsRetainMemResEnabled false, IsWriteProtectedInAS false, MemoryReserve 100
   VAR RETAIN
      OB82ErrorCounter : USInt;   // //Counter for error buffer
      CounterDiagStatusUpdate : USInt;   // //Counter for another error
      ErrorDataOB82 { S7_SetPoint := 'True'} : Array[1..200] of "stt_OB82";   // //buffer for error from OB82
   END_VAR
BEGIN
END_DATA_BLOCK

DATA_BLOCK "CONFIG_MODBUS_TCP_SERVER"   // DB87
TITLE = CONECT MODBUS TCP SERVER
{ S7_Optimized_Access := 'TRUE' }
AUTHOR : rtecmer
VERSION : 0.1
// stored: AutoNumber true, DBAccessibleFromOPCUA true, IsOnlyStoredInLoadMemory false, IsRetainMemResEnabled false, IsWriteProtectedInAS false, MemoryReserve 100
   VAR
      CONNECT_MODBUS_TCP_Serwer_1 { S7_SetPoint := 'True'} : TCON_IP_v4;
      ERROR_STATUS_SERWER_1 : Word;   // wartość błędu
      ERROR_STATUS_SERWER_2 : Word := 16#0;   // wartość błędu
      ERROR_STATUS_SERWER_3 : Word := 16#0;   // wartość błędu
      ERROR_STATUS_SERWER_4 : Word := 16#0;   // wartość błędu
      "CONFIG SERWER_1" : Struct
         STATUS { S7_SetPoint := 'True'} : Word;   // Status połączenia TCP Modbus
         error : Bool;   // błąd
         dr : Bool;   // dane czytane
         ndr : Bool;   // dane gotowe
      END_STRUCT;
      "CONFIG SERWER_2" : Struct
         STATUS { S7_SetPoint := 'True'} : Word;   // Status połączenia TCP Modbus
         error : Bool;   // błąd
         dr : Bool;   // dane czytane
         ndr : Bool;   // dane gotowe
      END_STRUCT;
      "CONFIG SERWER_3" : Struct
         STATUS { S7_SetPoint := 'True'} : Word;   // Status połączenia TCP Modbus
         error : Bool;   // błąd
         dr : Bool;   // dane czytane
         ndr : Bool;   // dane gotowe
      END_STRUCT;
      "CONFIG SERWER_4" : Struct
         STATUS { S7_SetPoint := 'True'} : Word;   // Status połączenia TCP Modbus
         error : Bool;   // błąd
         dr : Bool;   // dane czytane
         ndr : Bool;   // dane gotowe
      END_STRUCT;
      Time_Loop_modbustcp : Time;   // czas obiegu pętli modbus tcp
   END_VAR
BEGIN
   CONNECT_MODBUS_TCP_Serwer_1.InterfaceId := 64;
   CONNECT_MODBUS_TCP_Serwer_1.ID := 1;
   CONNECT_MODBUS_TCP_Serwer_1.ConnectionType := 11;
   CONNECT_MODBUS_TCP_Serwer_1.LocalPort := 502;
END_DATA_BLOCK

DATA_BLOCK "MB_TCP_CLIENT"   // DB86
TITLE = CONECT MODBUS TCP SERVER
{ S7_Optimized_Access := 'FALSE' }
AUTHOR : rtecmer
VERSION : 0.1
// stored: AutoNumber true, DBAccessibleFromOPCUA true, IsOnlyStoredInLoadMemory false, IsWriteProtectedInAS false
   VAR
      MB_Client_Receiving : Struct
         Input : Struct
            req : Bool;
            disconnect : Bool;
            mode : USInt;
            mbDataAddr : UDInt;
            CONNECT_ID : UInt := 2;
            IP_OCTET_1 : USInt;
            IP_OCTET_2 : USInt := 0;
            IP_OCTET_3 : USInt := 0;
            IP_OCTET_4 : USInt := 0;
            IP_PORT : UInt;
            MB_MODE : USInt;
            MB_DATA_ADDR : UDInt;
            DATA_LEN : UInt;
            PORT : UInt;
            InOut : Struct
               done : Bool;
               busy : Bool;
               error : Bool;
               STATUS : Word;
               ERROR_STATUS : Word;
            END_STRUCT;
         END_STRUCT;
         tagsStep : Struct
            "step" : Byte;
         END_STRUCT;
      END_STRUCT;
      MB_Client_Receiving_Time : Struct   // Pobieranie nastaw godzin
         Input : Struct
            req : Bool;
            disconnect : Bool;
            mode : USInt;
            mbDataAddr : UDInt;
            CONNECT_ID : UInt := 2;
            IP_OCTET_1 : USInt;
            IP_OCTET_2 : USInt := 0;
            IP_OCTET_3 : USInt := 0;
            IP_OCTET_4 : USInt := 0;
            IP_PORT : UInt;
            MB_MODE : USInt;
            MB_DATA_ADDR : UDInt;
            DATA_LEN : UInt;
            PORT : UInt;
            InOut : Struct
               done : Bool;
               busy : Bool;
               error : Bool;
               STATUS : Word;
               ERROR_STATUS : Word;
            END_STRUCT;
         END_STRUCT;
         tagsStep : Struct
            "step" : Byte;
         END_STRUCT;
      END_STRUCT;
      MB_Client_Sending : Struct   // instancja konfiguracji klient wysyłanie
         Input : Struct
            req : Bool;
            disconnect : Bool;
            mode : USInt;
            mbDataAddr : UDInt;
            CONNECT_ID : UInt;
            IP_OCTET_1 : USInt;
            IP_OCTET_2 : USInt := 0;
            IP_OCTET_3 : USInt := 0;
            IP_OCTET_4 : USInt := 0;
            IP_PORT : UInt;
            MB_MODE : USInt;
            MB_DATA_ADDR : UDInt;
            DATA_LEN : UInt;
            PORT : UInt;
            InOut : Struct
               done : Bool;
               busy : Bool;
               error : Bool;
               STATUS : Word;
               ERROR_STATUS : Word;
            END_STRUCT;
         END_STRUCT;
         tagsStep : Struct
            "step" : Byte;
         END_STRUCT;
      END_STRUCT;
      MB_Client_Sending_1 : Struct   // instancja konfiguracji klient wysyłanie
         Input : Struct
            req : Bool;
            disconnect : Bool;
            mode : USInt;
            mbDataAddr : UDInt;
            CONNECT_ID : UInt;
            IP_OCTET_1 : USInt;
            IP_OCTET_2 : USInt := 0;
            IP_OCTET_3 : USInt := 0;
            IP_OCTET_4 : USInt := 0;
            IP_PORT : UInt;
            MB_MODE : USInt;
            MB_DATA_ADDR : UDInt;
            DATA_LEN : UInt;
            PORT : UInt;
            InOut : Struct
               done : Bool;
               busy : Bool;
               set_step_17 { ExternalAccessible := 'False'; ExternalVisible := 'False'; ExternalWritable := 'False'} : Bool;   // bit inicjacji wysłąnia nowej wartości
               error : Bool;
               STATUS : Word;
               ERROR_STATUS : Word;
            END_STRUCT;
         END_STRUCT;
         tagsStep : Struct
            "step" : Byte;
         END_STRUCT;
      END_STRUCT;
      MB_Client_Sending_2 : Struct   // instancja konfiguracji klient wysyłanie
         Input : Struct
            req : Bool;
            disconnect : Bool;
            mode : USInt;
            mbDataAddr : UDInt;
            CONNECT_ID : UInt;
            IP_OCTET_1 : USInt;
            IP_OCTET_2 : USInt := 0;
            IP_OCTET_3 : USInt := 0;
            IP_OCTET_4 : USInt := 0;
            IP_PORT : UInt;
            MB_MODE : USInt;
            MB_DATA_ADDR : UDInt;
            DATA_LEN : UInt;
            PORT : UInt;
            InOut : Struct
               done : Bool;
               busy : Bool;
               error : Bool;
               STATUS : Word;
               ERROR_STATUS : Word;
            END_STRUCT;
         END_STRUCT;
         tagsStep : Struct
            "step" : Byte;
         END_STRUCT;
      END_STRUCT;
      MB_Client_Sending_3 : Struct   // instancja konfiguracji klient wysyłanie
         Input : Struct
            req : Bool;
            disconnect : Bool;
            mode : USInt;
            mbDataAddr : UDInt;
            CONNECT_ID : UInt;
            IP_OCTET_1 : USInt;
            IP_OCTET_2 : USInt := 0;
            IP_OCTET_3 : USInt := 0;
            IP_OCTET_4 : USInt := 0;
            IP_PORT : UInt;
            MB_MODE : USInt;
            MB_DATA_ADDR : UDInt;
            DATA_LEN : UInt;
            PORT : UInt;
            InOut : Struct
               done : Bool;
               busy : Bool;
               error : Bool;
               STATUS : Word;
               ERROR_STATUS : Word;
            END_STRUCT;
         END_STRUCT;
         tagsStep : Struct
            "step" : Byte;
         END_STRUCT;
      END_STRUCT;
      MB_Client_Sending_4 : Struct   // instancja konfiguracji klient wysyłanie
         Input : Struct
            req : Bool;
            disconnect : Bool;
            mode : USInt;
            mbDataAddr : UDInt;
            CONNECT_ID : UInt;
            IP_OCTET_1 : USInt;
            IP_OCTET_2 : USInt := 0;
            IP_OCTET_3 : USInt := 0;
            IP_OCTET_4 : USInt := 0;
            IP_PORT : UInt;
            MB_MODE : USInt;
            MB_DATA_ADDR : UDInt;
            DATA_LEN : UInt;
            PORT : UInt;
            InOut : Struct
               done : Bool;
               busy : Bool;
               error : Bool;
               STATUS : Word;
               ERROR_STATUS : Word;
            END_STRUCT;
         END_STRUCT;
         tagsStep : Struct
            "step" : Byte;
         END_STRUCT;
      END_STRUCT;
      MB_Client_Sending_5 : Struct   // instancja konfiguracji klient wysyłanie
         Input : Struct
            req : Bool;
            disconnect : Bool;
            mode : USInt;
            mbDataAddr : UDInt;
            CONNECT_ID : UInt;
            IP_OCTET_1 : USInt;
            IP_OCTET_2 : USInt := 0;
            IP_OCTET_3 : USInt := 0;
            IP_OCTET_4 : USInt := 0;
            IP_PORT : UInt;
            MB_MODE : USInt;
            MB_DATA_ADDR : UDInt;
            DATA_LEN : UInt;
            PORT : UInt;
            InOut : Struct
               done : Bool;
               busy : Bool;
               error : Bool;
               STATUS : Word;
               ERROR_STATUS : Word;
            END_STRUCT;
         END_STRUCT;
         tagsStep : Struct
            "step" : Byte;
         END_STRUCT;
      END_STRUCT;
      "step" : Byte;
   END_VAR
BEGIN
END_DATA_BLOCK

DATA_BLOCK "ModbusTCP_error"   // DB43
{ S7_Optimized_Access := 'TRUE' }
VERSION : 0.1
// stored: AutoNumber true, DBAccessibleFromOPCUA true, IsOnlyStoredInLoadMemory false, IsRetainMemResEnabled false, IsWriteProtectedInAS false, MemoryReserve 100
   VAR
      MB_Client_Sending_error_Code : Word;
      "step" : Byte;
   END_VAR
BEGIN
END_DATA_BLOCK

DATA_BLOCK "dbHoldRegSlave_to_MT101"   // DB100
{ S7_Optimized_Access := 'FALSE' }
VERSION : 0.1
// stored: AutoNumber false, DBAccessibleFromOPCUA true, IsOnlyStoredInLoadMemory false, IsWriteProtectedInAS false
   VAR
      Status_Sterowanie : Struct
         instvValveZ1 : Word := 33924;   // Zasuwa Status Z1
         instvValveZ2 : Word := 33924;   // Zasuwa Status Z2
         instvValveZ3 : Word := 33924;   // Zasuwa Status Z3
         instvValveZ4 : Word := 33924;   // Zasuwa Status Z4
         instvValveZ5 : Word := 33924;   // Zasuwa Status Z5
         instvValveZ6 : Word := 33924;   // Zasuwa Status Z6
         instvValveZ7 : Word := 33924;   // Zasuwa Status Z7
         instvValveZ8 : Word := 33924;   // Zasuwa Status Z8
         instvValveZ9 : Word := 33924;   // Zasuwa Status Z9
         instvValveZ10 : Word := 33924;   // Zasuwa Status Z10
         instControllDrivers_1 : Int;   // Bity sterowania napędami (start, stop, otwórz, zamknij) / Bity sterowania napędami (start, stop, otwórz, zamknij) Pompami M1-M4, Zasuwami Z1, Z2, Z3, Z4
         instControllDrivers_2 : Int;   // Bity przełączenia trybu pracy napędów / Bity sterowania napędami ( otwórz, zamknij, start, stop) Zasuwami Z5, Z6, Z7, Z8, Z9, Z10, Z11, Z12
         instConrol_ManAut_1 : Int;   // Bity przełączenia trybu pracy napędów / Bity przełączenia trybu pracy napędów M1-M4, Zasuwami Z1, Z2, Z3, Z4
         instConrol_ManAut_2 : Int;   // Bity przełączenia trybu pracy napędów / Bity przełączenia trybu pracy napędów Z5, Z6, Z7, Z8, Z9, Z10, Z11, Z12
         instLevelTank1 : Int;   // Poziom zbiornik
         instLevelTank2 : Int;   // Poziom zbiornik
         instLevelTank3 : Int;   // Poziom zbiornik
         instLevelTank4 : Int;   // Poziom zbiornik
         instPosition_Z10 : Real;   // rezerwa / Zadawanie położenia Z10
         instClearFault1 : Int;   // Bity kasowania alarmów napędów M1-M4, Z1 - Z12
         instSygSter_1 : Int;   // rezerwa / Sygnały sterowania strategią pompownia - 0= wyłaczone, 1=dosilanie, 2=przetłaczanie,3=automat, 4=ręczne
         instSygSter_2 : Int;   // Sygnały sterowania cyklem zbiorniki 0-wyłączone, 1=dobowy, 2=tygodniowy, 3=ręczne
         instCurrent_Inverter : Int;   // Aktualny prądu falownika
         instHz_Inverter : Int;   // Aktualne Hz na falowniku
      END_STRUCT;
      Pomiary : Struct
         instLevelSetFilling : Real;   // Zadany poziom napełniania
         instLevelSetEmptying : Real;   // Zadany poziom opróżniania
         instSetbarDN225_B6 : Real;   // Zadany ciśnienie tłóczenia kierunek miasto, Modbus 40035
         instSetbarDN500_B5 : Real;   // Zadana ciśnienie dosilania kierunek dosilanie "0" Modbus 40037
         instSetBarMinB9 : Real;   // Zadawana dolna granica ciśnienia studnia "Granica" Modbus 40039
         instB5bar_act : Real;   // Aktualne ciśnienie zasilania z sieci
         instPozitionZ10_act : Real;   // Aktualna pozycja zasuwy Z10
         instFlowDN500_act : Real;   // Przepływ DN500 (l/s) aktualny, zasilanie zbiorników, DOSILANIE, Modbus 40055
         instFlowDN500_sum : Real;   // SUMA przepływu Dolna DN500 Modbus 40057
      END_STRUCT;
      Godziny : Struct
         instHourStart_Filling : Int;   // Godzina start napełniania
         instMinutStart_Filling : Int;   // Minuta start napełniania
         instHourStop_Filling : Int;   // Godzina stop napełniania
         instMinutStopt_Filling : Int;   // Minuta stop napełniania
         instHourStart_City : Int;   // Godzina start przetłaczanie miasto DN225
         instMinutStart_City : Int;   // Minuty start przetłaczanie miasto DN225
         instHourStop_City : Int;   // Godzina stop przetłaczanie miasto DN225
         instMinutStopt_City : Int;   // Minuty stop przetłaczanie miasto DN225
         instHourStart_Replen : Int;   // Godzina start przetłaczanie magistrala DN500
         instMinutStart_Replen : Int;   // Minuty start przetłaczanie magistrala DN500
         instHourStop_Replen : Int;   // Godzina stop przetłaczanie magistrala DN500
         instMinutStopt_Replen : Int;   // Minuty stop przetłaczanie magistrala DN500
      END_STRUCT;
   END_VAR
BEGIN
END_DATA_BLOCK

DATA_BLOCK "dbHold_Sending"   // DB57
TITLE = Instancja danych serwera TCP
{ S7_Optimized_Access := 'FALSE' }
AUTHOR : rtecmer
VERSION : 0.1
// Instancja do przechowywania danych dla funkcji Modbus TCP - Blok danych przesyłanych do PLC Pompownia
// stored: AutoNumber true, DBAccessibleFromOPCUA true, IsOnlyStoredInLoadMemory false, IsWriteProtectedInAS false
   VAR
      data : Struct
         actB5_bar_magistrala : Real;   // 4001-4002 Pomiar ciśnienia magistrala - dosilanie
         act_poziom_ZB1 : Real;   // 4003-4004 Pomiar poziom w zbiorniku
         act_poziom_ZB2 : Real;   // 4005-4006 Pomiar poziom w zbiorniku
         act_poziom_ZB3 : Real;   // 4007-4008 Pomiar poziom w zbiorniku
         act_poziom_ZB4 : Real;   // 4009-4010 Pomiar poziom w zbiorniku
         act_przepływ_VF_Q2 : Real;   // 4011-4012 Aktualny przepływ VF
         "act_przepływ-VR_Q2" : Real;   // 4013-4014 Aktualny przepływ VR wsteczny
         sum_przepływ_Q2 : Real;   // 4015-4016
         stat : Struct
            status_Z1 : Word;   // 4017
            status_Z2 : Word;   // 4018
            status_Z3 : Word;   // 4019
            status_Z4 : Word;   // 4020
            status_Z5 : Word;   // 4021
            status_Z6 : Word;   // 4022
            status_Z7 : Word;   // 4023
            status_Z8 : Word;   // 4024
            status_Z9 : Word;   // 4025
            status_Z10 : Word;   // 4026
            status_przepływomierz_Q2 : Word;   // 4027 status przepływomierza DN500
            act_położenie_Z10 : Word;   // 4028 Położenie zasuwy Z10 [%]
            komunikacja_PLC : Word;   // 4029 Kontrola komunikacji PLC1 - PLC2 wartość 0 wysyłane do PLC1
            control : Struct
               set_poziom_napełniania : Real;   // 4030 - 4031 wartość zadana poziomu napełniania
               set_poziom_opróżniania : Real;   // 4032 - 4033 wartość zadana poziomu opróżniania
               control_2 : Struct
                  set_res_bity_sterowania_napęami_1 : Word;   // 4034 bity sterowania napędami
                  set_res_bity_sterowania_napęami_2 : Word;   // 4035 bity sterowania napędami
                  set_res_bity_tryb_napędów_1 : Word;   // 4036 bity sterowania przełączaniem trybów pracy
                  set_res_bity_tryb_napędów_2 : Word;   // 4037 bity sterowania przełączaniem trybów pracy
                  rez_alarm_napędów : Word;   // 4038 bity kasowania alarmów napędów
                  set_strategia_sterowania : Word;   // 4039 (Bit 53.0 - Wyłączony), (Bit 53.1 - Dosilanie), (Bit 53.2 - Przetłączanie), (Bit 53.3 - Automat), (Bit 53.4 - Ręczne )
                  set_sterowanie_cyklem : Word;   // 4040 (Bit 55.0 - Cykl wyłączony (Bit 55.1 - Cykl dobowy), (Bit 55.2 - Cykl tygodniowy), (Bit 55.3 - Cykl ręczny)
                  set_położenie_Z10 : Word;   // 4041Położenie zasuwy Z10 [%]
                  komunikacjaPLC : Word;   // 4042 kontrola komunikacji wysyłanie -> 0
               END_STRUCT;
            END_STRUCT;
         END_STRUCT;
         "Time" : Struct
            start_napełnianie : DTL;
            Stop_napełnianie : DTL;
            Start_przetłaczanie_1 : DTL;
            Stop_przetłaczanie_1 : DTL;
            Start_dosilanie_1 : DTL;
            Stop_dosilanie_1 : DTL;
         END_STRUCT;
      END_STRUCT;
   END_VAR
BEGIN
END_DATA_BLOCK

DATA_BLOCK "dbHold_download"   // DB58
TITLE = Instancja danych serwera TCP
{ S7_Optimized_Access := 'FALSE' }
AUTHOR : rtecmer
VERSION : 0.1
// Instancja dla funkcji Modbus TCP. Blok danych przechowujący dane pobrane z PLC Pompownia (zadane )
// stored: AutoNumber false, DBAccessibleFromOPCUA true, IsOnlyStoredInLoadMemory false, IsWriteProtectedInAS false
   VAR
      sterowanie : Struct
         act_położenie_Z10 : Word;   // Położenie zasuwy Z10 [%]
         set_poziom_napełniania : Real;   // wartość zadana poziomu napełniania
         set_poziom_opróżniania : Real;   // wartość zadana poziomu opróżniania
         set_res_bity_sterowania_napęami_1 : Word;   // bity sterowania napędami
         set_res_bity_sterowania_napęami_2 : Word := 16#0;   // bity sterowania napędami
         set_res_bity_tryb_napędów_1 : Word;   // bity sterowania przełączaniem trybów pracy
         set_res_bity_tryb_napędów_2 : Word := 16#0;   // bity sterowania przełączaniem trybów pracy
         rez_alarm_napędów : Word;   // bity kasowania alarmów napędów
         set_strategia_sterowania : Word;   // 0 - wyłączone, 1- Dosilanie, 2- Przetłaczanie, 3 - Automat
         set_sterowanie_cyklem : Word;   // 0- wyłączone, 1-Dobowe, 2- Tygodniowe, 3- Ręczne
         set_położenie_Z10 : Word;   // Położenie zasuwy Z10 [%]
         komunikacjaPLC : Word;   // kontrola komunikacji wysyłanie -PLC2 - PLC1
         set_magistrala_alarm_min_bar : Real;   // ciśnienie alarmu awaria na magistrali B5
      END_STRUCT;
      SendingTimes : Struct
         start_napełnianie : DTL;
         Stop_napełnianie : DTL;
         Start_przetłaczanie_1 : DTL;
         Stop_przetłaczanie_1 : DTL;
         Start_dosilanie_1 : DTL;
         Stop_dosilanie_1 : DTL;
      END_STRUCT;
   END_VAR
BEGIN
END_DATA_BLOCK

DATA_BLOCK "tempdbHold_SendingTCP"   // DB6
{ S7_Optimized_Access := 'FALSE' }
VERSION : 0.1
// stored: AutoNumber true, DBAccessibleFromOPCUA true, IsOnlyStoredInLoadMemory false, IsWriteProtectedInAS false
   VAR
      sterowanie : Struct
         act_położenie_Z10 : Word;   // Położenie zasuwy Z10 [%]
         set_poziom_napełniania : Real;   // wartość zadana poziomu napełniania
         set_poziom_opróżniania : Real;   // wartość zadana poziomu opróżniania
         set_res_bity_sterowania_napęami_1 : Word;   // bity sterowania napędami
         set_res_bity_sterowania_napęami_2 : Word := 16#0;   // bity sterowania napędami
         set_res_bity_tryb_napędów_1 : Word;   // bity sterowania przełączaniem trybów pracy
         set_res_bity_tryb_napędów_2 : Word := 16#0;   // bity sterowania przełączaniem trybów pracy
         rez_alarm_napędów : Word;   // bity kasowania alarmów napędów
         set_strategia_sterowania : Word;   // 0 - wyłączone, 1- Dosilanie, 2- Przetłaczanie, 3 - Automat
         set_sterowanie_cyklem : Word;   // 0- wyłączone, 1-Dobowe, 2- Tygodniowe, 3- Ręczne
         set_położenie_Z10 : Word;   // Położenie zasuwy Z10 [%]
         komunikacjaPLC : Word;   // kontrola komunikacji wysyłanie -PLC2 - PLC1
      END_STRUCT;
      SendingTimes : Struct
         start_napełnianie : DTL;
         Stop_napełnianie : DTL;
         Start_przetłaczanie_1 : DTL;
         Stop_przetłaczanie_1 : DTL;
         Start_dosilanie_1 : DTL;
         Stop_dosilanie_1 : DTL;
      END_STRUCT;
      actB5_bar_magistrala : Real;   // 4001-4002 Pomiar ciśnienia magistrala - dosilanie
      act_poziom_ZB1 : Real;   // 4003-4004 Pomiar poziom w zbiorniku
      act_poziom_ZB2 : Real;   // 4005-4006 Pomiar poziom w zbiorniku
      act_poziom_ZB3 : Real;   // 4007-4008 Pomiar poziom w zbiorniku
      act_poziom_ZB4 : Real;   // 4009-4010 Pomiar poziom w zbiorniku
      act_przepływ_VF_Q2 : Real;   // 4011-4012 Aktualny przepływ VF
      "act_przepływ-VR_Q2" : Real;   // 4013-4014 Aktualny przepływ VR wsteczny
      sum_przepływ_Q2 : Real;   // 4015-4016
      status_Z1 : Word;   // 4017
      status_Z2 : Word;   // 4018
      status_Z3 : Word;   // 4019
      status_Z4 : Word;   // 4020
      status_Z5 : Word;   // 4021
      status_Z6 : Word;   // 4022
      status_Z7 : Word;   // 4023
      status_Z8 : Word;   // 4024
      status_Z9 : Word;   // 4025
      status_Z10 : Word;   // 4026
      status_przepływomierz_Q2 : Word;   // 4027 status przepływomierza DN500
      act_położenie_Z10 : Word;   // 4028 Położenie zasuwy Z10 [%]
      komunikacja_PLC : Word;   // 4029 Kontrola komunikacji PLC1 - PLC2 wartość 0 wysyłane do PLC1
      set_poziom_napełniania : Real;   // 4030 - 4031 wartość zadana poziomu napełniania
      set_poziom_opróżniania : Real;   // 4032 - 4033 wartość zadana poziomu opróżniania
      set_res_bity_sterowania_napęami_1 : Word;   // 4034 bity sterowania napędami
      set_res_bity_sterowania_napęami_2 : Word;   // 4035 bity sterowania napędami
      set_res_bity_tryb_napędów_1 : Word;   // 4036 bity sterowania przełączaniem trybów pracy
      set_res_bity_tryb_napędów_2 : Word;   // 4037 bity sterowania przełączaniem trybów pracy
      rez_alarm_napędów : Word;   // 4038 bity kasowania alarmów napędów
      set_strategia_sterowania : Word;   // 4039 (Bit 53.0 - Wyłączony), (Bit 53.1 - Dosilanie), (Bit 53.2 - Przetłączanie), (Bit 53.3 - Automat), (Bit 53.4 - Ręczne )
      set_sterowanie_cyklem : Word;   // 4040 (Bit 55.0 - Cykl wyłączony (Bit 55.1 - Cykl dobowy), (Bit 55.2 - Cykl tygodniowy), (Bit 55.3 - Cykl ręczny)
      set_położenie_Z10 : Word;   // 4041Położenie zasuwy Z10 [%]
      komunikacjaPLC : Word;   // 4042 kontrola komunikacji wysyłanie -> 0
      start_napełnianie : DTL;
      Stop_napełnianie : DTL;
      Start_przetłaczanie_1 : DTL;
      Stop_przetłaczanie_1 : DTL;
      Start_dosilanie_1 : DTL;
      Stop_dosilanie_1 : DTL;
   END_VAR
BEGIN
END_DATA_BLOCK

DATA_BLOCK "ERR_Enum"   // DB105
{ S7_Optimized_Access := 'TRUE' }
VERSION : 0.1
// stored: AutoNumber false, DBAccessibleFromOPCUA true, IsOnlyStoredInLoadMemory false, IsRetainMemResEnabled false, IsWriteProtectedInAS false, MemoryReserve 0
   VAR
      GetErrorID : Array[0..27] of Word;
      SoftwareError { S7_SetPoint := 'True'} : "stt_ERR_Enum_SoftwareError";
      OB80 : Array[0..5] of Byte;
   END_VAR
BEGIN
   GetErrorID[0] := 16#2503;
   GetErrorID[1] := 16#2520;
   GetErrorID[2] := 16#2522;
   GetErrorID[3] := 16#2523;
   GetErrorID[4] := 16#2524;
   GetErrorID[5] := 16#2525;
   GetErrorID[6] := 16#2528;
   GetErrorID[7] := 16#2529;
   GetErrorID[8] := 16#252C;
   GetErrorID[9] := 16#2530;
   GetErrorID[10] := 16#2533;
   GetErrorID[11] := 16#2538;
   GetErrorID[12] := 16#2539;
   GetErrorID[13] := 16#253A;
   GetErrorID[14] := 16#253C;
   GetErrorID[15] := 16#253D;
   GetErrorID[16] := 16#253E;
   GetErrorID[17] := 16#253F;
   GetErrorID[18] := 16#2550;
   GetErrorID[19] := 16#2551;
   GetErrorID[20] := 16#2575;
   GetErrorID[21] := 16#2576;
   GetErrorID[22] := 16#2577;
   GetErrorID[23] := 16#25A0;
   GetErrorID[24] := 16#25A1;
   GetErrorID[25] := 16#25A2;
   GetErrorID[26] := 16#2942;
   GetErrorID[27] := 16#2943;
END_DATA_BLOCK

DATA_BLOCK "ERR_ErrorBufferFull"   // DB106
{ S7_Optimized_Access := 'TRUE' }
VERSION : 0.1
// stored: AutoNumber false, DBAccessibleFromOPCUA true, IsOnlyStoredInLoadMemory false, IsRetainMemResEnabled false, IsWriteProtectedInAS false, MemoryReserve 0
   VAR
      Error { S7_SetPoint := 'True'} : ErrorStruct;
   END_VAR
   VAR RETAIN
      SoftwareError { S7_SetPoint := 'True'} : Array[0..4] of "stt_ERR_SoftwareError";
      GetError { S7_SetPoint := 'True'} : Array[0..27] of "stt_ERR_GetError";
      CounterDiagStatusUpdate : UInt;
   END_VAR
BEGIN
END_DATA_BLOCK

DATA_BLOCK "ERR_ErrorOB"   // DB107
{ S7_Optimized_Access := 'TRUE' }
VERSION : 0.1
// stored: AutoNumber false, DBAccessibleFromOPCUA true, IsOnlyStoredInLoadMemory false, IsRetainMemResEnabled false, IsWriteProtectedInAS false, MemoryReserve 0
   VAR RETAIN
      OB80 { S7_SetPoint := 'True'} : Array[0..5] of "stt_ERR_OB80";
   END_VAR
BEGIN
END_DATA_BLOCK

DATA_BLOCK "V_ErrorOB"   // DB108
{ S7_Optimized_Access := 'TRUE' }
VERSION : 0.1
// stored: AutoNumber false, DBAccessibleFromOPCUA true, IsOnlyStoredInLoadMemory false, IsRetainMemResEnabled false, IsWriteProtectedInAS false, MemoryReserve 0
   VAR
      StartUp { S7_SetPoint := 'True'} : "stt_ERR_StartUpOB";   // //Error read in OB100
      OB80 : Bool;   // //Executed OB80 Time error interrupt
      ResetErrorOB : Bool;   // //Variable connected with button in web site
   END_VAR
BEGIN
END_DATA_BLOCK

DATA_BLOCK "V_SoftwareError"   // DB109
{ S7_Optimized_Access := 'TRUE' }
VERSION : 0.1
// stored: AutoNumber false, DBAccessibleFromOPCUA true, IsOnlyStoredInLoadMemory false, IsRetainMemResEnabled false, IsWriteProtectedInAS false, MemoryReserve 0
   VAR
      SoftwareFunctions : Bool;   // //Error is appear in called function
      GetErrorFunction : Bool;   // //Function GET_ERROR() return error
      DiagnosticBuffer : Bool;   // //Error is appear in diagnostic buffer
      ResetErrorSoftware : Bool;   // //Variable connected with button in web site
   END_VAR
BEGIN
END_DATA_BLOCK

DATA_BLOCK "V_LED"   // DB110
{ S7_Optimized_Access := 'TRUE' }
VERSION : 0.1
// stored: AutoNumber false, DBAccessibleFromOPCUA true, IsOnlyStoredInLoadMemory false, IsRetainMemResEnabled false, IsWriteProtectedInAS false, MemoryReserve 0
   VAR
      LED : Array[1..6] of Int;   // //Status for each module LED
   END_VAR
BEGIN
END_DATA_BLOCK

